# B&R Automation Studio project NAELD004C00R10L518F00 (part 43)

#### Act_Link.st
```iecst
(** 2021-05-18 **)
ACTION Act_Link:

	//ProdRcp
	bFollowerInfo	:= tyFollowerToLeaderTag.bProdWidthErr OR bProdRcpErrNotExist OR bProdRcpErrWidthMismatch;

	bLeaderInfo		:= (tyLeaderToFollowerTag.bProdWidthUSWarn OR tyLeaderToFollowerTag.bProdWidthDSWarn
	OR ((tyLeaderToFollowerTag.bProdNameUSWarn OR tyLeaderToFollowerTag.bProdNameDSWarn)
	AND (p_bAWPrep = TRUE) AND (p_bAWDis = FALSE) AND (p_eAWStat<>AWActGoWidthOff)));

	//Info Message
	IF bFollowerInfo THEN
		IF tyFollowerToLeaderTag.bProdWidthErr = TRUE OR bProdRcpErrWidthMismatch THEN

			p_sInfoMsg		:= 'Product Recipe Width Does Not Match';
			p_sInfoMsg		:= CONCAT(p_sInfoMsg , '$r$n');
			p_sInfoMsg		:= CONCAT(p_sInfoMsg , 'Check Product Width And');
			p_sInfoMsg		:= CONCAT(p_sInfoMsg , '$r$n');
			p_sInfoMsg		:= CONCAT(p_sInfoMsg , 'Leader Request Width');

		ELSIF bProdRcpErrNotExist THEN

			p_sInfoMsg		:= 'New Product Not Found';
			p_sInfoMsg		:= CONCAT(p_sInfoMsg , '$r$n');
			p_sInfoMsg		:= CONCAT(p_sInfoMsg , 'In Product Recipe List');
			p_sInfoMsg		:= CONCAT(p_sInfoMsg , '$r$n');
			p_sInfoMsg		:= CONCAT(p_sInfoMsg , 'Create New Product');
			p_sInfoMsg		:= CONCAT(p_sInfoMsg , '$r$n');
			p_sInfoMsg		:= CONCAT(p_sInfoMsg , 'In Product Setting');
		END_IF
	ELSE

		IF (tyLeaderToFollowerTag.sReqProdRcpNm<>p_tyCurrProdRcp.sRcpNm) AND (tyLeaderToFollowerTag.sReqProdRcpNm<>'')
			AND bLeaderInfo=FALSE THEN

			p_sInfoMsg		:= 'Leader Request New Recipe';
			p_sInfoMsg		:= CONCAT(p_sInfoMsg , '$r$n');
			p_sInfoMsg		:= CONCAT(p_sInfoMsg , 'Old Recipe Name : ');
			p_sInfoMsg		:= CONCAT(p_sInfoMsg , p_tyDispProdRcp.sRcpNm);
			p_sInfoMsg		:= CONCAT(p_sInfoMsg , '$r$n');
			p_sInfoMsg		:= CONCAT(p_sInfoMsg , 'Old Recipe Width : ');
			sWidthInUMTemp	:= DINT_TO_STRING(p_tyDispProdRcp.diWidthInUM / 1000);
			p_sInfoMsg		:= CONCAT(p_sInfoMsg , sWidthInUMTemp);
			p_sInfoMsg		:= CONCAT(p_sInfoMsg , '$r$n');
			p_sInfoMsg		:= CONCAT(p_sInfoMsg , 'New Recipe Name : ');
			p_sInfoMsg		:= CONCAT(p_sInfoMsg , tyLeaderToFollowerTag.sReqProdRcpNm);
			p_sInfoMsg		:= CONCAT(p_sInfoMsg , '$r$n');
			p_sInfoMsg		:= CONCAT(p_sInfoMsg , 'New Recipe Width : ');
			sWidthInUMTemp	:= DINT_TO_STRING(tyLeaderToFollowerTag.diReqProdRcpWidth / 1000);
			p_sInfoMsg		:= CONCAT(p_sInfoMsg , sWidthInUMTemp);

		ELSIF tyLeaderToFollowerTag.bProdNameUSWarn THEN
			p_sInfoMsg		:= 'US Machine Request New Recipe';
			p_sInfoMsg		:= CONCAT(p_sInfoMsg , '$r$n');
			p_sInfoMsg		:= CONCAT(p_sInfoMsg , 'Old Recipe Name : ');
			p_sInfoMsg		:= CONCAT(p_sInfoMsg , p_tyDispProdRcp.sRcpNm);
			p_sInfoMsg		:= CONCAT(p_sInfoMsg , '$r$n');
			p_sInfoMsg		:= CONCAT(p_sInfoMsg , 'Old Recipe Width : ');
			sWidthInUMTemp	:= DINT_TO_STRING(p_tyDispProdRcp.diWidthInUM / 1000); //Modify 18052021
			p_sInfoMsg		:= CONCAT(p_sInfoMsg , sWidthInUMTemp);
			p_sInfoMsg		:= CONCAT(p_sInfoMsg , '$r$n');
			p_sInfoMsg		:= CONCAT(p_sInfoMsg , 'New Recipe Name : ');
			p_sInfoMsg		:= CONCAT(p_sInfoMsg , tyLeaderToFollowerTag.sReqProdRcpNm);
			p_sInfoMsg		:= CONCAT(p_sInfoMsg , '$r$n');
			p_sInfoMsg		:= CONCAT(p_sInfoMsg , 'New Recipe Width : ');
			sWidthInUMTemp	:= DINT_TO_STRING(tyLeaderToFollowerTag.diReqProdRcpWidth / 1000);
			p_sInfoMsg		:= CONCAT(p_sInfoMsg , sWidthInUMTemp);

		ELSIF tyLeaderToFollowerTag.bProdNameDSWarn THEN
			p_sInfoMsg		:= 'Different Recipe';
			p_sInfoMsg		:= CONCAT(p_sInfoMsg , '$r$n');
			p_sInfoMsg		:= CONCAT(p_sInfoMsg , 'From DS Machine');
			p_sInfoMsg		:= CONCAT(p_sInfoMsg , '$r$n');
			p_sInfoMsg		:= CONCAT(p_sInfoMsg , 'Current Recipe Name : ');
			p_sInfoMsg		:= CONCAT(p_sInfoMsg , p_tyCurrProdRcp.sRcpNm);
			p_sInfoMsg		:= CONCAT(p_sInfoMsg , '$r$n');
			p_sInfoMsg		:= CONCAT(p_sInfoMsg , 'Current Recipe Width : ');
			sWidthInUMTemp	:= DINT_TO_STRING(p_tyCurrProdRcp.diWidthInUM2 / 1000);
			p_sInfoMsg		:= CONCAT(p_sInfoMsg , sWidthInUMTemp);

		ELSIF tyLeaderToFollowerTag.bProdWidthUSWarn THEN
			p_sInfoMsg		:= 'Product Recipe Width Does Not Match';
			p_sInfoMsg		:= CONCAT(p_sInfoMsg , '$r$n');
			p_sInfoMsg		:= CONCAT(p_sInfoMsg , 'Check Product Width And');
			p_sInfoMsg		:= CONCAT(p_sInfoMsg , '$r$n');
			p_sInfoMsg		:= CONCAT(p_sInfoMsg , 'Leader Request Width');

		ELSIF tyLeaderToFollowerTag.bProdWidthDSWarn THEN
			p_sInfoMsg		:= 'Same Recipe : ';
			p_sInfoMsg		:= CONCAT(p_sInfoMsg , p_tyDispProdRcp.sRcpNm);
			p_sInfoMsg		:= CONCAT(p_sInfoMsg , '$r$n');
			p_sInfoMsg		:= CONCAT(p_sInfoMsg , 'But Different Width');
			p_sInfoMsg		:= CONCAT(p_sInfoMsg , '$r$n');
			p_sInfoMsg		:= CONCAT(p_sInfoMsg , 'With DS Machine');
			p_sInfoMsg		:= CONCAT(p_sInfoMsg , '$r$n');
			p_sInfoMsg		:= CONCAT(p_sInfoMsg , 'Machine Outgoing Width : ');
			sWidthInUMTemp	:= DINT_TO_STRING(p_tyDispProdRcp.diWidthInUM2 / 1000);
			p_sInfoMsg		:= CONCAT(p_sInfoMsg , sWidthInUMTemp);

		END_IF
	END_IF

	//Accept New Recipe Condition (Before Loaded New Recipe)
	IF p_eLinkNtParamProjMag = LDMagDual OR p_eLinkNtParamProjMag = LDMagTriple  THEN
		p_bAccNewRcpCond	:= (p_bLinkOpsRun = TRUE)  AND (p_bLinkConvHvBrd = FALSE);
	END_IF

	//Update New Recipe Condition (After Loaded New Recipe)
	p_bUpdtNewRcpCond	:= TRUE;

	//Recipe Different
	//p_bInternalReqProdRcpDiff	:= memcmp(ADR(p_tyCurrProdRcp) , ADR(p_tyInternalReqProdRcp) , SIZEOF(p_tyCurrProdRcp)) <> 0;
	//p_bUpdtProdRcpDiff			:= memcmp(ADR(p_tyCurrProdRcp) , ADR(tyUpdtProdRcp) , SIZEOF(p_tyCurrProdRcp)) <> 0;
	//p_bRlsBrdProdRcpDiff		:= memcmp(ADR(p_tyCurrProdRcp) , ADR(tyRlsBrdProdRcpNm) , SIZEOF(p_tyCurrProdRcp)) <> 0;

	IF p_bErr THEN
		eCurrMachineStat := InError;
	ELSE
		IF p_bWarning THEN
			eCurrMachineStat := Warning;
		ELSE
			IF p_bOps THEN
				eCurrMachineStat := Run;
			ELSE
				IF p_bManual THEN
					eCurrMachineStat := Manual;
				ELSE
					eCurrMachineStat := Stop;
				END_IF
			END_IF
		END_IF
	END_IF

END_ACTION
```

#### Act_LinkEn.st
```iecst
(** 2019-04-26 **)
ACTION Act_LinkEn:

	//Link bPrep, bEn & bDis
	IF p_bLinkNtParamProjLaneBPrep = FALSE THEN
		p_bDis	:= (p_bLinkStartupRun = TRUE) OR (p_eLinkMcParamDSACommMod = McSetCommModHermes);
	ELSE
		p_bDis	:= (p_bLinkStartupRun = TRUE) OR (p_eLinkMcParamDSACommMod = McSetCommModHermes) OR (p_eLinkMcParamDSBCommMod = McSetCommModHermes);
	END_IF

END_ACTION
```

### LCS.typ
```iecst
(*2019-07-10*)
(**)
(*Action*)

TYPE
	eLCSAction :
		(
		LCSActIdle := 0,
		LCSActAddProd := 1,
		LCSActAddMultiProd := 2,
		LCSActEditProd := 3,
		LCSActEditMultiProd := 4,
		LCSActOverWriteProd := 5,
		LCSActOverWriteMultiProd := 6,
		LCSActDelProd := 7,
		LCSActDelMultiProd := 8,
		LCSActRunProd := 9,
		LCSActUploadProd := 10,
		LCSActUploadMultiProd := 11
		);
END_TYPE

(**)
(*Data*)

TYPE
	eLCSOpsStatus :
		(
		LCSOpsStatusAuto,
		LCSOpsStatusManual,
		LCSOpsStatusStop,
		LCSOpsStatusError,
		LCSOpsStatusWarning
		);
	tyLCSTagNm : 	STRUCT
		eAct : eLCSAction;
		eStat : eLCSAction;
		udiStatus : UDINT;
		sErrMsg : STRING[200];
		iIdxAct : INT;
		iIdxStat : INT;
		tyProdRcpInfo : tyProdRcpParam;
		tyCurrProdRcpParam : tyProdRcpParam;
		sCurrRcpNm : STRING[30];
		rCurrWidth : REAL;
		eCurrOpsStatus : eLCSOpsStatus;
		usiBrdStatus : USINT;
		usiMode : USINT;
		iTopToBtm : INT;
		sLastModified : STRING[80];
		bMngRcpEn : BOOL;
		bLiveData : BOOL;
		bLFEn : BOOL;
		sMcAlmMsg : STRING[255];
		bSectionLeaderEn : BOOL;
	END_STRUCT;
END_TYPE
```

### LCSLF.var
```iecst
(*2019-06-12*)
(**)
(*Action & State & Status*)
VAR
	p_LCSLFStat : UDINT;
	p_LCSLFStatus : UDINT;
	p_LCSLFStatTxt : UDINT;
END_VAR
(**)
(*Alarm*)
VAR
	p_LCSLFAlmData : UDINT;
	p_LCSLFInfoData : UDINT;
END_VAR
(**)
(*Output*)
VAR
	p_LCSLF_PLCStatus : UDINT;
	p_LCSLFChkLmt : UDINT;
	p_LCSLFAccDataMnl : UDINT;
	p_LCSLFUpdtDataMnl : UDINT;
	p_LCSLFUpdtProdRcpNm : UDINT;
	p_LCSLFUpdtProdWidth : UDINT;
	p_LCSLFMagAccOrder : UDINT;
	p_LCSLFMagOrderPos : UDINT;
END_VAR
```

### Program Logical/LCS/LCS

#### InputRef_Link.var
```iecst
(*2019-04-24*)
(**)
VAR
	p_bLinkStartupRun : REFERENCE TO BOOL;
	p_bLinkNtParamLCSLFPrep : REFERENCE TO BOOL;
	p_bLinkNtParamLCSManageRcpPrep : REFERENCE TO BOOL;
	p_bLinkNtParamLCSReqRcpPrep : REFERENCE TO BOOL;
	p_bLinkNtParamLCSLiveDatPrep : REFERENCE TO BOOL;
	p_bLinkMcParamLCSLFEn : REFERENCE TO BOOL;
	p_bLinkMcParamLCSManageRcpEn : REFERENCE TO BOOL;
	p_bLinkMcParamLCSReqRcpEn : REFERENCE TO BOOL;
	p_bLinkMcParamLCSLiveDatEn : REFERENCE TO BOOL;
END_VAR
(**)
VAR
	p_bLinkNtParamProjLaneBPrep : REFERENCE TO BOOL;
	p_tyLinkMcParamMagParamSelected : REFERENCE TO tyMagRcpParam;
END_VAR
(**)
VAR
	p_eLinkNtParamProjMag : REFERENCE TO eLDMag;
	p_bLinkPullConvHvBrd : REFERENCE TO BOOL;
	p_bLinkBffr1MagRemoved : REFERENCE TO BOOL;
	p_bLinkBffr2MagRemoved : REFERENCE TO BOOL;
	p_bLinkBffr3MagRemoved : REFERENCE TO BOOL;
END_VAR
```

#### Local.var
```iecst
(*2019-06-12*)
(**)
(*Local Action, State & Status*)
(**)
(*Local Alarm*)
VAR
	a_tyAlmText : ARRAY[10000..10099] OF tyAlmTxt := [(sAlmText:='LCS Disable'),(sAlmText:='LCS Manage Recipe Disabled'),(sAlmText:='LCS Leader Follower Disabled'),7(0),(sAlmText:='Out Of Range While Accepting New Recipe'),(sAlmText:='Out Of Range While Managing Product'),(sAlmText:='Recipe Name Empty While Adding Product'),(sAlmText:='Recipe List Full While Adding Product'),(sAlmText:='Recipe Name Exist While Adding Product'),(sAlmText:='Recipe Program Error While Adding Product'),(sAlmText:='Check Limit Error While Adding Multiple Product'),(sAlmText:='Recipe Name Empty While Adding Multiple Product'),(sAlmText:='Recipe List Full While Adding Multiple Product'),(sAlmText:='Recipe Name Exist While Adding Multiple Product'),(sAlmText:='Recipe Program Error While Adding Multiple Product'),(sAlmText:='Check Limit Error While Editing Product'),(sAlmText:='Recipe Name Empty While Editing Product'),(sAlmText:='Recipe Name Not Exist While Editing Product'),(sAlmText:='Recipe Program Error While Editing Product'),(sAlmText:='Check Limit Error While Editing Multiple Product'),(sAlmText:='Recipe Name Empty While Editing Multiple Product'),(sAlmText:='Recipe Name Not Exist While Editing Multiple Product'),(sAlmText:='Recipe Program Error While Editing Multiple Product'),(sAlmText:='Check Limit Error While Overwriting Product'),(sAlmText:='Recipe Name Empty While Overwriting Product'),(sAlmText:='Recipe List Full While Overwriting Product'),(sAlmText:='Recipe Program Error While Overwriting Product'),(sAlmText:='Check Limit Error While Overwriting Multiple Product'),(sAlmText:='Recipe Name Empty While Overwriting Multiple Product'),(sAlmText:='Recipe List Full While Overwriting Multiple Product'),(sAlmText:='Recipe Program Error While Overwriting Multiple Product'),(sAlmText:='Check Limit Error While Deleting Product'),(sAlmText:='Recipe Name Empty While Deleting Product'),(sAlmText:='Recipe Name Not Exist While Deleting Product'),(sAlmText:='Recipe Program Error While Deleting Product'),(sAlmText:='Check Limit Error While Deleting Multiple Product'),(sAlmText:='Recipe Name Empty While Deleting Multiple Product'),(sAlmText:='Recipe Name Not Exist While Deleting Multiple Product'),(sAlmText:='Recipe Program Error While Deleting Multiple Product'),(sAlmText:='Recipe Name Empty While Uploading Product'),(sAlmText:='Recipe Name Not Exist While Uploading Product'),(sAlmText:='Recipe Program Error While Uploading Product'),(sAlmText:='Get Recipe Info Error While Editing Product'),(sAlmText:='Local Recipe Is Latest Compare With LCS Recipe While Editing Product'),(sAlmText:='Local Recipe Is Latest Compare With LCS Recipe While Editing Multiple Product'),(sAlmText:='Get Recipe Info Error While Editing Multiple Product'),48(0)];
END_VAR
(**)
(*Local Output*)
VAR
	eLCSMngRcp_LCSAct : eLCSAction;
	iLCSMngRcp_LCSIdxAct : INT;
	iLCSMngRcp_LCSIdxStat : INT;
	tyLCSMngRcp_LCSProdRcpInfo : tyProdRcpParam;
	eLCSLF_LCSAct : eLCSAction;
	tyLCSLF_LCSProdRcpInfo : tyProdRcpParam;
	bChkLmtOK : BOOL;
	bChkLmtNG : BOOL;
END_VAR
(**)
(*Local Input*)
VAR
	bPrep : BOOL := TRUE;
	bEn : BOOL := TRUE;
	bDis : BOOL := FALSE;
	eLCSMngRcp_PLCStat : eLCSAction;
	udiLCSMngRcp_PLCStatus : UDINT;
	iLCSMngRcp_PLCIdxAct : INT;
	iLCSMngRcp_PLCIdxStat : INT;
	tyLCSMngRcp_PLCProdRcpInfo : tyProdRcpParam;
	eLCSLF_PLCStat : eLCSAction;
	udiLCSLF_PLCStatus : UDINT;
	bLCSMngRcpChkLmt : BOOL;
	bLCSLFChkLmt : BOOL;
	bOpsRun : BOOL;
	bError : BOOL;
	bWarning : BOOL;
	bInfo : BOOL;
	bUIManual : BOOL;
	tyProdRcpCurrRcp : tyProdRcpParam;
	tyNtParamCurr : tyNtParam;
	sProgNm : STRING[15] := 'LCS';
	bNtSettingsLoadDone : BOOL := TRUE;
END_VAR
(**)
(*Local*)
VAR
	bInitDone : BOOL;
	bInitialDone : BOOL;
	tyTagNm : tyLCSTagNm;
	bLFRun : BOOL;
	bMngRcpRun : BOOL;
	sLastModifiedTemp : STRING[80];
	sAddMsg : STRING[80];
END_VAR
```

#### Act_Background.st
```iecst
(** 2019-05-21 **)
ACTION Act_Background:

	Act_Background_LiveData;

END_ACTION
```

#### Act_InitGlobal.st
```iecst
(** 2019-06-12 **)
ACTION Act_InitGlobal:

	(* Always Change If Project Change *)

	//Pass Data To Link
	p_bLinkStartupRun ACCESS p_StartupRun;
	p_bLinkNtParamLCSLFPrep ACCESS p_NtParamLCSLFPrep;
	p_bLinkNtParamLCSManageRcpPrep ACCESS p_NtParamLCSManageRcpPrep;
	p_bLinkNtParamLCSReqRcpPrep ACCESS p_NtParamLCSReqRcpPrep;
	p_bLinkNtParamLCSLiveDatPrep ACCESS p_NtParamLCSLiveDatPrep;
	p_bLinkMcParamLCSLFEn ACCESS p_McParamLCSLFEn;
	p_bLinkMcParamLCSManageRcpEn ACCESS p_McParamLCSManageRcpEn;
	p_bLinkMcParamLCSReqRcpEn ACCESS p_McParamLCSReqRcpEn;
	p_bLinkMcParamLCSLiveDatEn ACCESS p_McParamLCSLiveDatEn;

	p_bLinkNtParamProjLaneBPrep ACCESS p_NtParamProjLaneBPrep;
	p_tyLinkMcParamMagParamSelected ACCESS p_MagRcpCurrRcp;

	p_eLinkNtParamProjMag ACCESS p_NtParamProjMag;
	p_bLinkPullConvHvBrd ACCESS p_PullConvHvBrd;
	p_bLinkBffr1MagRemoved ACCESS p_Buffer1MagRemoved;
	p_bLinkBffr2MagRemoved ACCESS p_Buffer2MagRemoved;
	p_bLinkBffr3MagRemoved ACCESS p_Buffer3MagRemoved;

	//Pass Data To Internal Use
	p_eLCSMngRcp_PLCStat ACCESS p_LCSMngRcpStat;
	p_udiLCSMngRcp_PLCStatus ACCESS p_LCSMngRcp_PLCStatus;
	p_iLCSMngRcp_PLCIdxAct ACCESS p_LCSMngRcp_PLCIdxAct;
	p_iLCSMngRcp_PLCIdxStat ACCESS p_LCSMngRcp_PLCIdxStat;
	p_tyLCSMngRcp_PLCProdRcpInfo ACCESS p_LCSMngRcp_PLCProdRcpInfo;
	p_eLCSLF_PLCStat ACCESS p_LCSLFStat;
	p_udiLCSLF_PLCStatus ACCESS p_LCSLF_PLCStatus;
	p_bLCSMngRcpChkLmt ACCESS p_LCSMngRcpChkLmt;
	p_bLCSLFChkLmt ACCESS p_LCSLFChkLmt;
	p_bOpsRun ACCESS p_OpsRun;
	p_bError ACCESS p_AlarmErr;
	p_bWarning ACCESS p_AlarmWarning;
	p_bInfo ACCESS p_AlarmInfo;
	p_bUIManual ACCESS p_UIUIMnlMod;
	p_tyProdRcpCurrRcp ACCESS p_Follower2UpdtProdRcp;	//Assign With Conveyor Last Zone (Live Data Update)
	p_tyNtParamCurr ACCESS p_NtParamCurr;
	p_sProgNm ACCESS p_NtParamLCSProgNm;
	p_bNtSettingsLoadDone ACCESS p_StartupNtSettingsLoadDone;

	(* Always Change If Project Change *)

END_ACTION
```

#### Act_Link.st
```iecst
(** 2019-07-15 **)
ACTION Act_Link:

	//Check Limit
	IF p_bLCSMngRcpChkLmt OR p_bLCSLFChkLmt THEN

		IF tyTagNm.tyProdRcpInfo.sRcpNm = '' THEN

			bChkLmtOK	:= FALSE;
			bChkLmtNG	:= TRUE;
			sAddMsg		:= 'Recipe Name Empty ';

		ELSIF tyTagNm.tyProdRcpInfo.diWidthInUM < p_tyNtParamCurr.tyProdRcpWidth.diMin THEN

			bChkLmtOK	:= FALSE;
			bChkLmtNG	:= TRUE;
			sAddMsg		:= 'Width Lower Limit ';

		ELSIF tyTagNm.tyProdRcpInfo.diWidthInUM > p_tyNtParamCurr.tyProdRcpWidth.diMax THEN

			bChkLmtOK	:= FALSE;
			bChkLmtNG	:= TRUE;
			sAddMsg		:= 'Width Upper Limit ';

		ELSIF NOT p_bLinkNtParamProjLaneBPrep AND (tyTagNm.tyProdRcpInfo.usiMcMod < DINT_TO_USINT(p_tyNtParamCurr.tyProdRcpMcModA.diMin)) THEN

			bChkLmtOK	:= FALSE;
			bChkLmtNG	:= TRUE;
			sAddMsg		:= 'Machine Mode Lower Limit ';

		ELSIF NOT p_bLinkNtParamProjLaneBPrep AND (tyTagNm.tyProdRcpInfo.usiMcMod > DINT_TO_USINT(p_tyNtParamCurr.tyProdRcpMcModA.diMax)) THEN

			bChkLmtOK	:= FALSE;
			bChkLmtNG	:= TRUE;
			sAddMsg		:= 'Machine Mode Upper Limit ';

		ELSIF p_bLinkNtParamProjLaneBPrep AND (tyTagNm.tyProdRcpInfo.usiMcMod < DINT_TO_USINT(p_tyNtParamCurr.tyProdRcpMcModAB.diMin)) THEN

			bChkLmtOK	:= FALSE;
			bChkLmtNG	:= TRUE;
			sAddMsg		:= 'Machine Mode Lower Limit ';

		ELSIF p_bLinkNtParamProjLaneBPrep AND (tyTagNm.tyProdRcpInfo.usiMcMod > DINT_TO_USINT(p_tyNtParamCurr.tyProdRcpMcModAB.diMax)) THEN

			bChkLmtOK	:= FALSE;
			bChkLmtNG	:= TRUE;
			sAddMsg		:= 'Machine Mode Upper Limit ';

		ELSIF tyTagNm.tyProdRcpInfo.diMaxSltValue < tyTagNm.tyProdRcpInfo.diMinSltValue THEN

			bChkLmtOK	:= FALSE;
			bChkLmtNG	:= TRUE;
			sAddMsg		:= 'Max Slot Lower Limit ';

		ELSIF tyTagNm.tyProdRcpInfo.diMaxSltValue > p_tyLinkMcParamMagParamSelected.diTtlSlt THEN

			bChkLmtOK	:= FALSE;
			bChkLmtNG	:= TRUE;
			sAddMsg		:= 'Max Slot Upper Limit ';

		ELSIF tyTagNm.tyProdRcpInfo.diMinSltValue < p_tyNtParamCurr.diProjMagMinSlt THEN

			bChkLmtOK	:= FALSE;
			bChkLmtNG	:= TRUE;
			sAddMsg		:= 'Min Slot Lower Limit ';

		ELSIF tyTagNm.tyProdRcpInfo.diMinSltValue > tyTagNm.tyProdRcpInfo.diMaxSltValue THEN

			bChkLmtOK	:= FALSE;
			bChkLmtNG	:= TRUE;
			sAddMsg		:= 'Min Slot Upper Limit ';

		ELSIF tyTagNm.tyProdRcpInfo.diPitch < p_tyNtParamCurr.tyProdRcpPitch.diMin THEN

			bChkLmtOK	:= FALSE;
			bChkLmtNG	:= TRUE;
			sAddMsg		:= 'Pitch Lower Limit ';

		ELSIF tyTagNm.tyProdRcpInfo.diPitch > (tyTagNm.tyProdRcpInfo.diMaxSltValue - tyTagNm.tyProdRcpInfo.diMinSltValue + 1) THEN

			bChkLmtOK	:= FALSE;
			bChkLmtNG	:= TRUE;
			sAddMsg		:= 'Pitch Upper Limit ';

		ELSIF LEN(tyTagNm.tyProdRcpInfo.sRcpNm) > 30 THEN

			bChkLmtOK	:= FALSE;
			bChkLmtNG	:= TRUE;
			sAddMsg		:= 'Recipe Name Length ';

		ELSE

			bChkLmtOK	:= TRUE;
			bChkLmtNG	:= FALSE;
			sAddMsg		:= '';

		END_IF

	ELSE

		bChkLmtOK	:= FALSE;
		bChkLmtNG	:= FALSE;

	END_IF

	//Update LCS Enable
	tyTagNm.bMngRcpEn		:= p_bLinkNtParamLCSManageRcpPrep AND p_bLinkMcParamLCSManageRcpEn;
	tyTagNm.bLFEn			:= p_bLinkNtParamLCSLFPrep AND p_bLinkMcParamLCSLFEn;
	tyTagNm.bLiveData		:= p_bLinkNtParamLCSLiveDatPrep AND p_bLinkMcParamLCSLiveDatEn;

	//tyTagNm.usiBrdStatus = 0 (Machine Empty)
	//tyTagNm.usiBrdStatus = 1 (Machine Not Empty)
	IF p_eLinkNtParamProjMag = LDMagDual THEN
		tyTagNm.usiBrdStatus	:= BOOL_TO_USINT(NOT(p_bLinkPullConvHvBrd = FALSE AND p_bLinkBffr1MagRemoved = TRUE AND p_bLinkBffr2MagRemoved = TRUE));
	ELSIF p_eLinkNtParamProjMag = LDMagTriple THEN
		tyTagNm.usiBrdStatus	:= BOOL_TO_USINT(NOT(p_bLinkPullConvHvBrd = FALSE AND p_bLinkBffr1MagRemoved = TRUE AND p_bLinkBffr2MagRemoved = TRUE AND p_bLinkBffr3MagRemoved = TRUE));
	END_IF

	//Action
	IF tyTagNm.eAct = LCSActRunProd THEN

		bLFRun		:= TRUE;
		bMngRcpRun	:= FALSE;

	ELSIF (tyTagNm.eAct = LCSActAddProd)
		OR (tyTagNm.eAct = LCSActAddMultiProd)
		OR (tyTagNm.eAct = LCSActEditProd)
		OR (tyTagNm.eAct = LCSActEditMultiProd)
		OR (tyTagNm.eAct = LCSActOverWriteProd)
		OR (tyTagNm.eAct = LCSActOverWriteMultiProd)
		OR (tyTagNm.eAct = LCSActDelProd)
		OR (tyTagNm.eAct = LCSActDelMultiProd)
		OR (tyTagNm.eAct = LCSActUploadProd)
		OR (tyTagNm.eAct = LCSActUploadMultiProd) THEN

		bLFRun		:= FALSE;
		bMngRcpRun	:= TRUE;

	ELSIF tyTagNm.eAct = LCSActIdle THEN

		bLFRun		:= FALSE;
		bMngRcpRun	:= FALSE;

	END_IF

	IF bLFRun = TRUE THEN
		eLCSLF_LCSAct			:= tyTagNm.eAct;
		tyLCSLF_LCSProdRcpInfo	:= tyTagNm.tyProdRcpInfo;

		tyLCSLF_LCSProdRcpInfo.bTopToBtm	:= INT_TO_BOOL(tyTagNm.iTopToBtm);

		sLastModifiedTemp	:= CONCAT('DT#' , tyTagNm.sLastModified);
		tyLCSLF_LCSProdRcpInfo.dtLastModified	:= STRING_TO_DT(sLastModifiedTemp);

		tyTagNm.eStat		:= p_eLCSLF_PLCStat;
		tyTagNm.udiStatus	:= p_udiLCSLF_PLCStatus;

		IF tyTagNm.udiStatus > 0 AND tyTagNm.udiStatus < 65534 THEN
			tyTagNm.sErrMsg	:= a_tyAlmText[tyTagNm.udiStatus].sAlmText;

			IF tyTagNm.udiStatus = 10010 OR tyTagNm.udiStatus = 10011 THEN
				tyTagNm.sErrMsg	:= CONCAT(sAddMsg , tyTagNm.sErrMsg);
			END_IF
		END_IF

	ELSIF bMngRcpRun = TRUE THEN
		eLCSMngRcp_LCSAct	:= tyTagNm.eAct;

		tyTagNm.eStat		:= p_eLCSMngRcp_PLCStat;
		tyTagNm.udiStatus	:= p_udiLCSMngRcp_PLCStatus;

		IF tyTagNm.udiStatus > 0 AND tyTagNm.udiStatus < 65534 THEN
			tyTagNm.sErrMsg	:= a_tyAlmText[tyTagNm.udiStatus].sAlmText;

			IF tyTagNm.udiStatus = 10010 OR tyTagNm.udiStatus = 10011 THEN
				tyTagNm.sErrMsg	:= CONCAT(sAddMsg , tyTagNm.sErrMsg);
			END_IF
		END_IF

		IF tyTagNm.eAct = LCSActUploadProd THEN
			IF tyTagNm.udiStatus = 0 THEN
				tyTagNm.tyProdRcpInfo	:= p_tyLCSMngRcp_PLCProdRcpInfo;

				tyTagNm.iTopToBtm	:= BOOL_TO_INT(tyLCSMngRcp_LCSProdRcpInfo.bTopToBtm);

				tyTagNm.sLastModified	:= DT_TO_STRING(tyLCSMngRcp_LCSProdRcpInfo.dtLastModified);
				tyTagNm.sLastModified	:= RIGHT(tyTagNm.sLastModified , (LEN(tyTagNm.sLastModified) - 3));

			ELSE
				tyLCSMngRcp_LCSProdRcpInfo	:= tyTagNm.tyProdRcpInfo;

				tyLCSMngRcp_LCSProdRcpInfo.bTopToBtm	:= INT_TO_BOOL(tyTagNm.iTopToBtm);
				tyLCSMngRcp_LCSProdRcpInfo.diWidthInUM2 := tyTagNm.tyProdRcpInfo.diWidthInUM;

				sLastModifiedTemp	:= CONCAT('DT#' , tyTagNm.sLastModified);
				tyLCSMngRcp_LCSProdRcpInfo.dtLastModified	:= STRING_TO_DT(sLastModifiedTemp);

			END_IF

		ELSIF tyTagNm.eAct = LCSActUploadMultiProd THEN
			iLCSMngRcp_LCSIdxStat	:= tyTagNm.iIdxAct;

			tyTagNm.iIdxStat		:= p_iLCSMngRcp_PLCIdxAct;

			tyTagNm.tyProdRcpInfo	:= p_tyLCSMngRcp_PLCProdRcpInfo;

			tyTagNm.iTopToBtm	:= BOOL_TO_INT(tyLCSMngRcp_LCSProdRcpInfo.bTopToBtm);

			tyTagNm.sLastModified	:= DT_TO_STRING(tyLCSMngRcp_LCSProdRcpInfo.dtLastModified);
			tyTagNm.sLastModified	:= RIGHT(tyTagNm.sLastModified , (LEN(tyTagNm.sLastModified) - 3));

		ELSE
			iLCSMngRcp_LCSIdxAct		:= tyTagNm.iIdxAct;
			tyLCSMngRcp_LCSProdRcpInfo	:= tyTagNm.tyProdRcpInfo;

			tyLCSMngRcp_LCSProdRcpInfo.bTopToBtm	:= INT_TO_BOOL(tyTagNm.iTopToBtm);
			tyLCSMngRcp_LCSProdRcpInfo.diWidthInUM2 := tyTagNm.tyProdRcpInfo.diWidthInUM;

			sLastModifiedTemp	:= CONCAT('DT#' , tyTagNm.sLastModified);
			tyLCSMngRcp_LCSProdRcpInfo.dtLastModified	:= STRING_TO_DT(sLastModifiedTemp);

			tyTagNm.iIdxStat	:= p_iLCSMngRcp_PLCIdxStat;

		END_IF

	ELSE

		eLCSLF_LCSAct		:= LCSActIdle;
		eLCSMngRcp_LCSAct	:= LCSActIdle;
		tyTagNm.eStat		:= LCSActIdle;
		tyTagNm.udiStatus	:= 65534;
		tyTagNm.sErrMsg		:= '';

	END_IF

END_ACTION
```

#### Init.st
```iecst
(** 2019-04-24 **)
PROGRAM _INIT

	(* Always Change If Project Change *)

	//Pass Address To Global Address For External Use
	//Action, State & Status

	//Alarm

	//Output
	p_LCS_LCSMngRcp_LCSAct			:= ADR(eLCSMngRcp_LCSAct);
	p_LCS_LCSMngRcp_LCSIdxAct		:= ADR(iLCSMngRcp_LCSIdxAct);
	p_LCS_LCSMngRcp_LCSIdxStat		:= ADR(iLCSMngRcp_LCSIdxStat);
	p_LCS_LCSMngRcp_LCSProdRcpInfo	:= ADR(tyLCSMngRcp_LCSProdRcpInfo);
	p_LCS_LCSLF_LCSAct				:= ADR(eLCSLF_LCSAct);
	p_LCS_LCSLF_LCSProdRcpInfo		:= ADR(tyLCSLF_LCSProdRcpInfo);
	p_LCSChkLmtOK					:= ADR(bChkLmtOK);
	p_LCSChkLmtNG					:= ADR(bChkLmtNG);
	p_LCSSectionLeaderEn			:= ADR(tyTagNm.bSectionLeaderEn);

	(* Always Change If Project Change *)

END_PROGRAM
```

### Program Logical/LCS/LCSLF

#### InputRef_Link.var
```iecst
(*2019-04-24*)
(**)
VAR
	sWidthInUMTemp : STRING[80];
	p_bLinkStartupRun : REFERENCE TO BOOL;
END_VAR
(**)
VAR
	p_bLinkNtParamProjLaneBPrep : REFERENCE TO BOOL;
	p_eLinkMcParamDSACommMod : REFERENCE TO eMcSetCommMod;
	p_eLinkMcParamDSBCommMod : REFERENCE TO eMcSetCommMod;
END_VAR
(**)
VAR
	p_bLinkOpsRun : REFERENCE TO BOOL;
	p_bLinkConvHvBrd : REFERENCE TO BOOL;
	p_bLinkOpsMagConvLD1QueryWO : REFERENCE TO BOOL;
	p_bLinkOpsMagConvLD2QueryWO : REFERENCE TO BOOL;
	p_bLinkOpsMagConvLD3QueryWO : REFERENCE TO BOOL;
	p_tyDTStructure : REFERENCE TO DTStructure;
	p_tyResponseFromMES1 : REFERENCE TO tyStatPlatformFromMES;
	p_tyResponseFromMES2 : REFERENCE TO tyStatPlatformFromMES;
	p_tyResponseFromMES3 : REFERENCE TO tyStatPlatformFromMES;
END_VAR
```

#### Local.var
```iecst
(*2019-06-28*)
(**)
(*Local Action, State & Status*)
VAR
	eAct : eLCSAction := LCSActIdle;
	eStat : eLCSAction := LCSActIdle;
	eStatus : eFBStatus := Idle;
	udiStatus : UDINT := 0;
	sStatTxt : STRING[200] := '';
	a_sStatText : ARRAY[0..50] OF STRING[200] := ['Idling','Adding Product','Adding Multiple Products','Editing Product','Editing Multiple Products','OverWrite Product','OverWrite Multiple Products','Deleting Product','Deleting Multiple Products','Running LCS Product','Uploading Product','Uploading Multiple Products',39('')];
END_VAR
(**)
(*Local Alarm*)
VAR
	tyAlmData : tyAlmDat;
	tyInfoData : tyAlmDat;
	a_tyAlmText : ARRAY[10000..10099] OF tyAlmTxt;
END_VAR
(**)
(*Local Output*)
VAR
	udiPLCStatus : UDINT;
	bChkLmt : BOOL;
	bAccDataMnl : BOOL;
	bUpdtDataMnl : BOOL;
	sUpdtProdRcpNm : STRING[30];
	diUpdtProdWidth : DINT;
END_VAR
(**)
(*Local Input*)
VAR
	udiRstErr : UDINT := 0;
	bPrep : BOOL := TRUE;
	bEn : BOOL := TRUE;
	bDis : BOOL := FALSE;
	tyCurrProdParam : tyProdRcpParam;
	bMnlAccData : BOOL;
	bAccData : BOOL;
	tyLCSProdRcpInfo : tyProdRcpParam;
	bChkLmtOK : BOOL;
	bChkLmtNG : BOOL;
	bAccNewRcpCond : BOOL;
	bUpdtNewRcpCond : BOOL;
	bAutoUpdtData : BOOL;
	bUIUpdtData : BOOL;
	sInfoMsg : STRING[200];
	sProgNm : STRING[15] := 'LCSLF';
	bNtSettingsLoadDone : BOOL := TRUE;
END_VAR
(**)
(*Local*)
VAR
	bRstErr : BOOL;
	udiRstErrOld : UDINT;
	bInitDone : BOOL;
	bInitialDone : BOOL;
	usiStep : USINT;
	usiProdUpdtDatStep : USINT;
	udiModuleNum : UDINT := 4101;
END_VAR
(*Local priority param*)
VAR
	bGUIDInserted : ARRAY[1..3] OF BOOL;
	a_MagGUID : ARRAY[1..3] OF STRING[80];
END_VAR
VAR RETAIN
	a_MagAccOrder : ARRAY[1..3] OF USINT; (*priority (output)*)
END_VAR
VAR
	usiMagPrior : ARRAY[1..3] OF USINT := [1,2,3];
	usiMagRun : ARRAY[1..3] OF USINT;
	usiSum : ARRAY[1..3] OF USINT;
	usiMagOrderPos : USINT;
	i : USINT;
	i1 : USINT;
	uiMilliSecOld : UINT;
END_VAR
```

#### Act_Alarm.st
```iecst
(** 2019-04-24 **)
ACTION Act_Alarm:

	//Error
	IF EDGEPOS(eStatus = Error) THEN

		tyAlmData.sProgNm		:= p_sProgNm;
		tyAlmData.udiCode		:= udiStatus;
		tyAlmData.eSeverity		:= AlmSeverityError;
		tyAlmData.udiRunTime	:= tyAlmData.udiRunTime + 1;
		tyAlmData.bAlm			:= TRUE;
		tyAlmData.udiModuleNum  := udiModuleNum;
		g_sLCSLFProgNm			:= p_sProgNm;

		//Get Error Message
		IF tyAlmData.udiCode < 10000 OR tyAlmData.udiCode > 10099 THEN
			tyAlmData.sAlmMsg	:= 'Unknown';
			tyAlmData.sRcyMsg	:= 'Unknown';
		ELSE
			tyAlmData.sAlmMsg	:= a_tyAlmText[tyAlmData.udiCode].sAlmText;
			tyAlmData.sRcyMsg	:= a_tyAlmText[tyAlmData.udiCode].sRcyText;
		END_IF

		sStatTxt	:= tyAlmData.sAlmMsg;

	ELSIF bRstErr AND (tyAlmData.udiCode <> 0) THEN

		tyAlmData.udiCode	:= 0;
		tyAlmData.eSeverity	:= AlmSeverityNA;
		tyAlmData.sAlmMsg	:= '';
		tyAlmData.sRcyMsg	:= '';
		tyAlmData.bAlm			:= FALSE;
		sStatTxt	:= a_sStatText[eStat];

	END_IF

END_ACTION
```

#### Act_InitGlobal.st
```iecst
(** 2019-05-07 **)
ACTION Act_InitGlobal:

	(* Always Change If Project Change *)

	//Pass Data To Link
	p_bLinkStartupRun ACCESS p_StartupRun;
	p_bLinkNtParamProjLaneBPrep ACCESS p_NtParamProjLaneBPrep;
	p_eLinkMcParamDSACommMod ACCESS p_McParamDSCommAMod;
	p_eLinkMcParamDSBCommMod ACCESS p_McParamDSCommBMod;

	p_bLinkOpsRun ACCESS p_OpsRun;
	p_bLinkConvHvBrd ACCESS p_PullConvHvBrd;
	p_bLinkOpsMagConvLD1QueryWO ACCESS p_OpsMagConvLD1QueryWO;
	p_bLinkOpsMagConvLD2QueryWO ACCESS p_OpsMagConvLD2QueryWO;
	p_bLinkOpsMagConvLD3QueryWO ACCESS p_OpsMagConvLD3QueryWO;
	p_tyDTStructure ACCESS p_TimeCurrDTStruct;
	p_tyResponseFromMES1 ACCESS p_TagFromMesMagConv1; //For we_fab
	p_tyResponseFromMES2 ACCESS p_TagFromMesMagConv2; //For we_fab
	p_tyResponseFromMES3 ACCESS p_TagFromMesMagConv3; //For we_fab

	//Pass Data To Internal Use
	p_eAct ACCESS p_LCS_LCSLF_LCSAct;
	p_udiRstErr ACCESS p_RstErrReset;
	p_bPrep ACCESS p_NtParamLCSLFPrep;
	p_bEn ACCESS p_McParamLCSLFEn;
	p_tyCurrProdParam ACCESS p_ProdRcpCurrRcp0;
	p_bMnlAccData ACCESS p_McParamMnlAccDat;
	p_bAccData ACCESS p_UIProdAccData;
	p_tyLCSProdRcpInfo ACCESS p_LCS_LCSLF_LCSProdRcpInfo;
	p_bChkLmtOK ACCESS p_LCSChkLmtOK;
	p_bChkLmtNG ACCESS p_LCSChkLmtNG;
	p_sProgNm ACCESS p_NtParamLCSLFProgNm;
	p_bNtSettingsLoadDone ACCESS p_StartupNtSettingsLoadDone;

	p_bUIBtnSectionLdr ACCESS P_UISectionLdr;
	p_bLCSSectionLeaderEn ACCESS p_LCSSectionLeaderEn;
	p_bMcParamSectionLdr ACCESS p_McParamSectionLeader;

	(* Always Change If Project Change *)

END_ACTION
```

#### Act_Link.st
```iecst
(** 2019-06-28 **)
ACTION Act_Link:

	p_sInfoMsg		:= 'LCS Request New Recipe';
	p_sInfoMsg		:= CONCAT(p_sInfoMsg , '$r$n');
	p_sInfoMsg		:= CONCAT(p_sInfoMsg , 'Old Recipe Name : ');
	p_sInfoMsg		:= CONCAT(p_sInfoMsg , p_tyCurrProdParam.sRcpNm);
	p_sInfoMsg		:= CONCAT(p_sInfoMsg , '$r$n');
	p_sInfoMsg		:= CONCAT(p_sInfoMsg , 'Old Recipe Width : ');
	sWidthInUMTemp	:= DINT_TO_STRING(p_tyCurrProdParam.diWidthInUM / 1000);
	p_sInfoMsg		:= CONCAT(p_sInfoMsg , sWidthInUMTemp);
	p_sInfoMsg		:= CONCAT(p_sInfoMsg , '$r$n');
	p_sInfoMsg		:= CONCAT(p_sInfoMsg , 'New Recipe Name : ');
	p_sInfoMsg		:= CONCAT(p_sInfoMsg , p_tyLCSProdRcpInfo.sRcpNm);
	p_sInfoMsg		:= CONCAT(p_sInfoMsg , '$r$n');
	p_sInfoMsg		:= CONCAT(p_sInfoMsg , 'New Recipe Width : ');
	sWidthInUMTemp	:= DINT_TO_STRING(p_tyLCSProdRcpInfo.diWidthInUM / 1000);
	p_sInfoMsg		:= CONCAT(p_sInfoMsg , sWidthInUMTemp);

	//Accept New Recipe Condition
	p_bAccNewRcpCond	:= p_bLinkOpsRun = TRUE AND p_bLinkConvHvBrd = FALSE;

	//@@@@@@@@@@@@@@@@@@@@@@@@@@@@@@@@@@@@@@@@@@@@@@@@@@@@@@@@@@@@@@@@@@@@@@
	//we_fabricate
//	IF  uiMilliSecOld <> p_tyDTStructure.millisec THEN
//		IF EDGEPOS(p_bLinkOpsMagConvLD1QueryWO) THEN //query false when rcp loaded
//			sMagazineId 		:= '1'; //Magazine position to mes
//			bGUIDInserted[1]	:= FALSE;
//			a_bQueryQueue[i2] 	:= TRUE;
//			i2 := i2 + 1;
//		ELSIF EDGEPOS(p_bLinkOpsMagConvLD2QueryWO) THEN
//			sMagazineId 		:= '2';
//			bGUIDInserted[2]	:= FALSE;
//			a_bQueryQueue[i2] 	:= TRUE;
//			i2 := i2 + 1;
//		ELSIF EDGEPOS(p_bLinkOpsMagConvLD3QueryWO) THEN
//			sMagazineId 		:= '3';
//			bGUIDInserted[3]	:= FALSE;
//			a_bQueryQueue[i2] 	:= TRUE;
//			i2 := i2 + 1;
//		END_IF
//	END_IF
	IF  uiMilliSecOld <> p_tyDTStructure.millisec THEN
		//Priority setting
		IF EDGEPOS(p_tyResponseFromMES1.iAcceptCondition >0)  OR EDGEPOS(p_tyResponseFromMES2.iAcceptCondition > 0)  OR EDGEPOS(p_tyResponseFromMES3.iAcceptCondition >0) THEN
			uiMilliSecOld :=  p_tyDTStructure.millisec;
			memset(ADR(usiSum),0,SIZEOF(usiSum));
			IF p_tyResponseFromMES1.iAcceptCondition >0 THEN
				usiSum[1] := 11;
			ELSIF p_tyResponseFromMES2.iAcceptCondition >0 THEN
				usiSum[2] := 12;
			ELSIF p_tyResponseFromMES3.iAcceptCondition >0 THEN
				usiSum[3] := 13;
			END_IF
		ELSE
			memset(ADR(usiSum),0,SIZEOF(usiSum));
		END_IF
	END_IF

//	FOR i := 1 TO 3 DO
//		usiSum[i]	:= usiSum[i] + usiMagPrior[i];
//		IF a_MagGUID[i] = tySendWorkOrderInfoRcv.tyData.sQueryId THEN
//			usiSum[i] := usiSum[i] + 10;
//		END_IF
//	END_FOR

	FOR i1:=1 TO 3 DO
		//Assign Magazine order
		IF  usiSum[i1] >=10 THEN
			IF a_MagAccOrder[1]=0 AND a_MagAccOrder[2]=0 AND a_MagAccOrder[3]=0 THEN
				a_MagAccOrder[i1] := 10; //output
				usiMagOrderPos := i1;
			ELSIF ((a_MagAccOrder[1]=0 AND a_MagAccOrder[2]=0) OR
				(a_MagAccOrder[2]=0 AND a_MagAccOrder[3]=0) OR
				(a_MagAccOrder[1]=0 AND a_MagAccOrder[3]=0)) AND a_MagAccOrder[i1] =0 THEN
				a_MagAccOrder[i1] := 20;
				usiMagOrderPos := i1;
			ELSIF (a_MagAccOrder[1]=0 OR a_MagAccOrder[2]=0 OR a_MagAccOrder[3]=0) AND a_MagAccOrder[i1] =0 THEN
				a_MagAccOrder[i1] := 30;
				usiMagOrderPos := i1;
			END_IF
			bGUIDInserted[i1] := FALSE;
		END_IF
	END_FOR

	//update magazine mmy
	IF a_MagAccOrder[1]<>0 AND a_MagAccOrder[2]<>0 AND a_MagAccOrder[3]<>0 THEN
	ELSIF a_MagAccOrder[1]<>10 AND a_MagAccOrder[2]<>10 AND a_MagAccOrder[3]<>10 THEN
		FOR i := 1 TO 3 DO
			IF a_MagAccOrder[i] <> 0 THEN
				a_MagAccOrder[i] := a_MagAccOrder[i] -10;
			END_IF
		END_FOR
	END_IF

END_ACTION
```

#### Act_LinkEn.st
```iecst
(** 2019-04-24 **)
ACTION Act_LinkEn:

	//Link bPrep, bEn & bDis
	IF p_bLinkNtParamProjLaneBPrep = FALSE THEN
		p_bDis	:= (p_bLinkStartupRun = TRUE) OR (p_eLinkMcParamDSACommMod = McSetCommModHermes);
	ELSE
		p_bDis	:= (p_bLinkStartupRun = TRUE) OR (p_eLinkMcParamDSACommMod = McSetCommModHermes) OR (p_eLinkMcParamDSBCommMod = McSetCommModHermes);
	END_IF

END_ACTION
```

#### Act_Main.st
```iecst
(** 2019-06-28 **)
ACTION Act_Main:

	//Main
	CASE eStat OF

		LCSActIdle:
			IF eStatus <> Idle THEN	//Reset Data
				//Private
				usiStep		:= 0;
				bAccDataMnl	:= FALSE;
				bChkLmt		:= FALSE;

				tyInfoData.sProgNm		:= '';
				tyInfoData.udiCode		:= 0;
				tyInfoData.eSeverity	:= AlmSeverityNA;
				tyInfoData.sAlmMsg		:= '';

				sStatTxt	:= a_sStatText[eStat];

			END_IF

			eStatus			:= Idle;
			udiPLCStatus	:= 65534;

		LCSActRunProd:
			IF eStatus = Idle OR eStatus = Busy THEN

				eStatus			:= Busy;
				udiPLCStatus	:= 65535;

				sStatTxt	:= a_sStatText[eStat];

				CASE usiStep OF
					0:
						//Check Limit
						bChkLmt	:= TRUE;

						IF p_bChkLmtOK = TRUE THEN
							usiStep			:= 1;
						ELSIF p_bChkLmtNG = TRUE THEN
							eStatus			:= Done;
							udiPLCStatus	:= 10010;	//Out Of Range While Accepting New Recipe
						END_IF

					1:
						//Manual Accept Data Check
						IF p_bMnlAccData = TRUE THEN
							bAccDataMnl	:= TRUE;

							//Info Message
							tyInfoData.sProgNm		:= p_sProgNm;
							tyInfoData.udiCode		:= 10000;
							tyInfoData.eSeverity	:= AlmSeverityInfo;
							tyInfoData.sAlmMsg		:= p_sInfoMsg;

							IF p_bAccData = TRUE THEN
								p_bAccData := FALSE; //2023_07_26_Debug for Manual Accept Data automatically accept after product change many times
								bAccDataMnl	:= FALSE;
								usiStep		:= 2;
							END_IF
						ELSE
							p_bAccData := FALSE; //2023_07_26_Debug for Manual Accept Data automatically accept after product change many times
							bAccDataMnl	:= FALSE;
							usiStep		:= 2;
						END_IF

					2:
						//Accept New Recipe Condition
						IF p_bAccNewRcpCond = TRUE THEN
							usiStep	:= 3;
						ELSE
							//Info Message
							tyInfoData.sProgNm		:= p_sProgNm;
							tyInfoData.udiCode		:= 10000;
							tyInfoData.eSeverity	:= AlmSeverityInfo;
							tyInfoData.sAlmMsg		:= p_sInfoMsg;
						END_IF

					3:
						//Accept New Recipe
						p_tyCurrProdParam	:= p_tyLCSProdRcpInfo;

						IF p_bLCSSectionLeaderEn = TRUE THEN
							p_bMcParamSectionLdr	:= TRUE;
							p_bUIBtnSectionLdr		:= TRUE;
						ELSE
							p_bMcParamSectionLdr	:= FALSE;
							p_bUIBtnSectionLdr		:= FALSE;

						END_IF

						usiStep	:= 4;

					4:
						//Clear Info Message
						tyInfoData.sProgNm		:= '';
						tyInfoData.udiCode		:= 0;
						tyInfoData.eSeverity	:= AlmSeverityNA;
						tyInfoData.sAlmMsg		:= '';

						usiStep	:= 0;

						eStatus			:= Done;
						udiPLCStatus	:= 0;

				END_CASE

			END_IF

		ELSE
			IF eStatus = Idle OR eStatus = Busy THEN
				eStatus	:= Done;
			END_IF

	END_CASE

END_ACTION
```

#### Init.st
```iecst
(** 2019-06-12 **)
PROGRAM _INIT

	(* Always Change If Project Change *)

	//Pass Address To Global Address For External Use
	//Action, State & Status
	p_LCSLFStat		:= ADR(eStat);
	p_LCSLFStatus	:= ADR(eStatus);
	p_LCSLFStatTxt	:= ADR(sStatTxt);

	//Alarm
	p_LCSLFAlmData	:= ADR(tyAlmData);
	p_LCSLFInfoData	:= ADR(tyInfoData);

	//Output
	p_LCSLF_PLCStatus		:= ADR(udiPLCStatus);
	p_LCSLFChkLmt			:= ADR(bChkLmt);
	p_LCSLFAccDataMnl		:= ADR(bAccDataMnl);
	p_LCSLFUpdtDataMnl		:= ADR(bUpdtDataMnl);
	p_LCSLFUpdtProdRcpNm	:= ADR(sUpdtProdRcpNm);
	p_LCSLFUpdtProdWidth	:= ADR(diUpdtProdWidth);

	p_LCSLFMagAccOrder 			:= ADR(a_MagAccOrder);
	p_LCSLFMagOrderPos 			:= ADR(usiMagOrderPos);

	(* Always Change If Project Change *)

END_PROGRAM
```

### Program Logical/LCS/LCSMngRcp

#### Act_Alarm.st
```iecst
(** 2019-04-24 **)
ACTION Act_Alarm:

	//Error
	IF EDGEPOS(eStatus = Error) THEN

		tyAlmData.sProgNm		:= p_sProgNm;
		tyAlmData.udiCode		:= udiStatus;
		tyAlmData.eSeverity		:= AlmSeverityError;
		tyAlmData.udiRunTime	:= tyAlmData.udiRunTime + 1;
		tyAlmData.bAlm			:= TRUE;
		tyAlmData.udiModuleNum  := udiModuleNum;
		g_sLCSMngRcpProgNm		:= p_sProgNm;

		//Get Error Message
		IF tyAlmData.udiCode < 10000 OR tyAlmData.udiCode > 10099 THEN
			tyAlmData.sAlmMsg	:= 'Unknown';
			tyAlmData.sRcyMsg	:= 'Unknown';
		ELSE
			tyAlmData.sAlmMsg	:= a_tyAlmText[tyAlmData.udiCode].sAlmText;
			tyAlmData.sRcyMsg	:= a_tyAlmText[tyAlmData.udiCode].sRcyText;
		END_IF

		sStatTxt	:= tyAlmData.sAlmMsg;

	ELSIF bRstErr AND (tyAlmData.udiCode <> 0) THEN

		tyAlmData.udiCode	:= 0;
		tyAlmData.eSeverity	:= AlmSeverityNA;
		tyAlmData.sAlmMsg	:= '';
		tyAlmData.sRcyMsg	:= '';
		tyAlmData.bAlm			:= FALSE;
		sStatTxt	:= a_sStatText[eStat];

	END_IF

END_ACTION
```

### Program Logical/Operations/Ops (IEC) - 1.00.0 - 

#### InputRef_Link.var
```iecst
(*2019-01-20*)
(**)
(*External*)
VAR
	p_bLinkOpsTravLifLDPaused : REFERENCE TO BOOL;
	p_bLinkOpsMagLD1Paused : REFERENCE TO BOOL;
	p_bLinkOpsMagLD2Paused : REFERENCE TO BOOL;
	p_bLinkOpsMagLD3Paused : REFERENCE TO BOOL;
	p_bLinkOpsMagLD4Paused : REFERENCE TO BOOL;
	p_bLinkOpsMagConvLD1Paused : REFERENCE TO BOOL;
	p_bLinkOpsMagConvLD2Paused : REFERENCE TO BOOL;
	p_bLinkOpsMagConvLD3Paused : REFERENCE TO BOOL;
	p_bLinkOpsMagConvLD4Paused : REFERENCE TO BOOL;
	p_bLinkUIOpsAct : REFERENCE TO eOperationsAction;
	p_bLinkSimuRun : REFERENCE TO BOOL;
	p_bLinkSimuStop : REFERENCE TO BOOL;
	p_bLinkOpsLifMagLDPaused : REFERENCE TO BOOL;
	p_bLinkProjLifterMagPlatform : REFERENCE TO BOOL;
END_VAR
```

#### Act_InitGlobal.st
```iecst
(** 2019-03-22 **)
ACTION Act_InitGlobal:

	(* Always Change If Project Change *)

	//Pass Data To Link
	p_bLinkOpsTravLifLDPaused ACCESS p_OpsTravLifLDPaused;
//	p_bLinkOpsMagLD1Paused ACCESS p_OpsMagLD1Paused;
//	p_bLinkOpsMagLD2Paused ACCESS p_OpsMagLD2Paused;
//	p_bLinkOpsMagLD3Paused ACCESS p_OpsMagLD3Paused;
//	p_bLinkOpsMagLD4Paused ACCESS p_OpsMagLD4Paused;
	p_bLinkOpsMagConvLD1Paused ACCESS p_OpsMagConvLD1Paused;
	p_bLinkOpsMagConvLD2Paused ACCESS p_OpsMagConvLD2Paused;
	p_bLinkOpsMagConvLD3Paused ACCESS p_OpsMagConvLD3Paused;
	p_bLinkOpsMagConvLD4Paused ACCESS p_OpsMagConvLD4Paused;
	p_bLinkUIOpsAct ACCESS p_UIOpsAct;
	p_bLinkSimuRun ACCESS p_SimuRun;
	p_bLinkSimuStop ACCESS p_SimuStop;

	p_bLinkProjLifterMagPlatform ACCESS p_NtParamProjLifterMagPlatform;
	p_bLinkOpsLifMagLDPaused ACCESS p_OpsLifMagLDPaused;

	//Pass Data To Internal Use
//	p_eAct ACCESS p_UIOpsAct;
	p_udiRstErr ACCESS p_RstErrReset;
	p_bNtSettingsLoadDone ACCESS p_StartupNtSettingsLoadDone;

	(* Always Change If Project Change *)

END_ACTION
```

#### Act_Link.st
```iecst
(** 2019-01-20 **)
ACTION Act_Link:

	IF p_bLinkProjLifterMagPlatform THEN

		p_bPaused	:= 	(p_bLinkOpsTravLifLDPaused AND p_bLinkOpsLifMagLDPaused);

	ELSE

		p_bPaused	:= 	(p_bLinkOpsTravLifLDPaused
	//					AND p_bLinkOpsMagLD1Paused AND p_bLinkOpsMagLD2Paused AND p_bLinkOpsMagLD3Paused AND p_bLinkOpsMagLD4Paused
						AND p_bLinkOpsMagConvLD1Paused AND p_bLinkOpsMagConvLD2Paused AND p_bLinkOpsMagConvLD3Paused  AND p_bLinkOpsMagConvLD4Paused);

	END_IF

END_ACTION
```

#### Act_LinkAction.st
```iecst
(** 2019-03-29 **)
ACTION Act_LinkAction:

	IF p_bLinkUIOpsAct <> OperationsActIdle THEN
		p_eAct ACCESS p_UIOpsAct;
	ELSIF EDGEPOS(p_bLinkSimuRun) THEN
		p_eAct := OperationsActStart;
	ELSIF EDGEPOS(p_bLinkSimuStop) THEN
		p_eAct := OperationsActStop;
	END_IF

	IF (eStat = OperationsActStart OR eStat = OperationsActStop) AND  eStatus = Done THEN
		eAct := OperationsActIdle;
		p_eAct := OperationsActIdle;
	END_IF

END_ACTION
```

#### Init.st
```iecst
(** 2019-04-16 **)
PROGRAM _INIT

	(* Always Change If Project Change *)

	//Pass Address To Global Address For External Use
	//Action, State & Status
	p_OpsStat		:= ADR(eStat);
	p_OpsStatus		:= ADR(eStatus);
	p_OpsStatTxt	:= ADR(sStatTxt);

	//Alarm

	//Output
	p_OpsOpsStatus			:= ADR(eOpsStatus);
	p_OpsStatusRun			:= ADR(bStatusRun);
	p_OpsStatusStop			:= ADR(bStatusStop);
	p_OpsStatusCycleStop	:= ADR(bStatusCycleStop);
	p_OpsStatusStep			:= ADR(bStatusStep);
	p_OpsRun				:= ADR(bRun);
	p_OpsStop				:= ADR(bStop);
	p_OpsStep				:= ADR(bStep);
	p_OpsPause				:= ADR(bPaused);
	(* Always Change If Project Change *)

END_PROGRAM
```

### OpsTravLifLD.typ - Do Not Change!!!
```iecst
(*2018-12-11*)
(**)
(*Configuration*)

TYPE
	eLDMod :
		(
		LDModLoadLnA,
		LDModLoadLnB,
		LDModLoadLnAB
		);
	eLDMag :
		(
		LDMagDual,
		LDMagTriple,
		LDMagQuadruple
		);
END_TYPE

(**)

TYPE
	tyParamTravLifLD : 	STRUCT
		a_bUSDis : ARRAY[1..4]OF BOOL := [4(FALSE)];
		a_bDSDis : ARRAY[1..4]OF BOOL := [4(FALSE)];
		a_usiUSPriority : ARRAY[1..4]OF USINT := [1,2,3,1(0)];
		a_usiDSPriority : ARRAY[1..4]OF USINT := [1,2,3,1(0)];
	END_STRUCT;
END_TYPE

(**)
(*Sequence*)

TYPE
	eTravLifLDStep :
		(
		TravLifLDStepNA,
		TravLifLDStepInitConv,
		TravLifLDStepInitInletPneuCls,
		TravLifLDStepInitInOutPneuCls,
		TravLifLDStepInitTravLif,
		TravLifLDStepInitAWTravLif,
		TravLifLDStepAWMov,
		TravLifLDStepTravLifMov,
		TravLifLDStepUSSigWait,
		TravLifLDStepUSSigRechk,
		TravLifLDStepInletPneuOpn,
		TravLifLDStepUSSigRechkTwice,
		TravLifLDStepUSComm,
		TravLifLDStepEntBrd,
		TravLifLDStepInletPneuCls,
		TravLifLDStepDSSigWait,
		TravLifLDStepDSSigRechk,
		TravLifLDStepOutletPneuOpn,
		TravLifLDStepDSSigRechkTwice,
		TravLifLDStepChkRgtSenForDBAOn,
		TravLifLDStepDSComm,
		TravLifLDStepExitBrd,
		TravLifLDStepOutletPneuCls,
		TravLifLDStepTranInErr
		);
	eTravLifLDStep1 :
		(
		TravLifLDStep1NA,
		TravLifLDStep1InitConv,
		TravLifLDStep1InitInletPneuCls,
		TravLifLDStep1InitInOutPneuCls,
		TravLifLDStep1InitTravLif,
		TravLifLDStep1InitAWTravLif,
		TravLifLDStep1DSSigWait100,
		TravLifLDStep1AWMov,
		TravLifLDStep1Standby,
		TravLifLDStep1USSigWait,
		TravLifLDStep1PreEntAllServo200,
		TravLifLDStep1PreEntMove300,
		TravLifLDStep1TraLifNxtUnlBffr,
		TravLifLDStep1PreEntTravLifMov,
		TravLifLDStep1EntTraLifMovRotCyl,
		TravLifLDStep1USSigRechk,
		TravLifLDStep1InletPneuOpn,
		MagPlat_Step1InletPneuOpn,
		TravLifLDStep1USSigRechkTwice,
		TravLifLDStep1USMagWidthChk,
		TravLifLDStep1USComm,
		TravLifLDStep1EntPullerExt,
		TravLifLDStep1EntPullerRetWait,
		TravLifLDStep1EntTravLifMov,
		TravLifLDStep1EntBrd,
		MagPlat_Step1EntBrd,
		TravLifLDStep1InletPneuCls,
		MagPlat_Step1InletPneuCls,
		TravLifLDStep1DSSigWait,
		TravLifLDStep1ExitTravLifMov,
		TravLifLDStep1InShutClsInt,
		TravLifLDStep1DSSigRechk,
		TravLifLDStep1OutletPneuOpn,
		TravLifLDStep1DSSigRechkTwice,
		TravLifLDStep1ChkRgtSenForDBAOn,
		TravLifLDStep1DSComm,
		TravLifLDStep1ExitBrd,
		TravLifLDStep1OutletPneuCls,
		TravLifLDStep1TranInErr,
		TravLifLDStep1TranOutBrdStuckErr,
		TravLifLDStep1MagWidthErr,
		TravLifLDStep1OutletShutErr,
		TravLifLDStep1ConvEntBrdLostErr
		);
	eTravLifLDPos :
		(
		TravLifLDPosInvalid,
		TravLifLDPosUS1,
		TravLifLDPosUS2,
		TravLifLDPosUS3,
		TravLifLDPosDS1,
		TravLifLDPosDS2,
		TravLifLDPosDS3,
		TravLifLDPosUS4
		);
END_TYPE
```

### OpsTravLifLD.var - Change By Project
```iecst
(*2019-03-25*)
(**)
(*Action & State & Status*)
(**)
(*Alarm*)
VAR
	p_OpsTravLifLDAlmData : UDINT;
END_VAR
(**)
(*Output*)
VAR
	p_OpsTravLifLDStepTxt : UDINT;
	p_OpsTravLifLDPaused : UDINT;
END_VAR
(**)
VAR
	p_OpsTravLifLDUSSMEMAAct1 : UDINT;
	p_OpsTravLifLDUSSMEMAAct2 : UDINT;
	p_OpsTravLifLDUSSMEMAAct3 : UDINT;
	p_OpsTravLifLDUSSMEMAAct4 : UDINT;
	p_OpsTravLifLDDSSMEMAAct1 : UDINT;
	p_OpsTravLifLDDSSMEMAAct2 : UDINT;
	p_OpsTravLifLDDSSMEMAAct3 : UDINT;
	p_OpsTravLifLDConvAct : UDINT;
	p_OpsTravLifLDAWAct : UDINT;
	p_OpsTravLifLDAWPushPullAct : UDINT;
	p_OpsTravLifLDTravAct : UDINT;
	p_OpsTravLifLDLifAct : UDINT;
	p_OpsTravLifLDInletPneuAct : UDINT;
	p_OpsTravLifLDInletPneuAct2 : UDINT;
	p_OpsTravLifLDInletPneuAct3 : UDINT;
	p_OpsTravLifLDOutletPneuAct : UDINT;
	p_OpsTravLifLDOutletPneuAct2 : UDINT;
	p_OpsTravLifLDPullerAct : UDINT;
END_VAR
(**)
VAR
	p_OpsTravLifLDPosGo : UDINT;
	p_OpsTravLifLDMagDis : UDINT;
	p_OpsTravLifLDGoUnloadSlt1 : UDINT;
	p_OpsTravLifLDGoUnloadSlt2 : UDINT;
	p_OpsTravLifLDGoUnloadSlt3 : UDINT;
	p_OpsTravLifLDGoUnloadSlt4 : UDINT;
	p_OpsTravLifLDInitConv : UDINT;
	p_OpsTravLifLDInitDone : UDINT;
	p_OpsTravLifLDUSComm : UDINT;
	p_OpsTravLifLDEntBrd : UDINT;
	p_OpsTravLifLDDSComm : UDINT;
	p_OpsTravLifLDExitBrd : UDINT;
	p_OpsTravLifLDAWPosDiff : UDINT;
	p_OpsTravLifULInDSPos : UDINT;
	p_OpsTravLifULUpdatePullSlot : UDINT;
	p_OpsTravLifLDBypCurtainSenCtrl : UDINT;
	p_OpsTravLifLBypCurtainWidthChg : UDINT;
	p_OpsTravLifLDBypCurtainLED : UDINT;
	p_OpsTravLifLDUSMagWidthChk : UDINT;
	p_OpsTravLifULTravGotoChkPt : UDINT;
	p_OpsTravLifWChkErrCmdUnclmp1 : UDINT;
	p_OpsTravLifWChkErrCmdUnclmp2 : UDINT;
	p_OpsTravLifWChkErrCmdUnclmp3 : UDINT;
	p_OpsTravLifMove : UDINT;
	p_OpsTravLifStandby : UDINT;
END_VAR
```

### Program Logical/Operations/OpsTravLifLD (IEC) - pne

#### InputRef.var
```iecst
(*2019-04-16*)
(**)
(*General*)
VAR
	p_udiRstErr : REFERENCE TO UDINT;
	p_bEn : REFERENCE TO BOOL;
	p_bDis : REFERENCE TO BOOL;
	p_bRun : REFERENCE TO BOOL;
	p_bStop : REFERENCE TO BOOL;
	p_bStep : REFERENCE TO BOOL;
	p_bGotoStandby : REFERENCE TO BOOL;
	p_bUnlockCover : REFERENCE TO BOOL;
END_VAR
(**)
(*Configuration*)
VAR
	p_sProgNm : REFERENCE TO STRING[15];
	p_bNtSettingsLoadDone : REFERENCE TO BOOL;
END_VAR
(**)
VAR
	p_eLDMod : REFERENCE TO eLDMod;
	p_eLDMag : REFERENCE TO eLDMag;
	p_bNonBffrMod : REFERENCE TO BOOL;
	p_bUSAllow : REFERENCE TO BOOL;
	p_bDSAllow : REFERENCE TO BOOL;
	p_bPullerRotCylPrep : REFERENCE TO BOOL;
	p_diPullerExtMaxSlt : REFERENCE TO DINT;
	p_diPullerExtMinSlt : REFERENCE TO DINT;
END_VAR
(**)
VAR
	p_bProdRcpCurrRcpTopToBtm : REFERENCE TO BOOL;
	p_diProdRcpCurrRcpPitch : REFERENCE TO DINT;
	p_diProdRcpCurrRcpPitchRear : REFERENCE TO DINT;
	p_diMinSlt : REFERENCE TO DINT;
	p_diMaxSlt : REFERENCE TO DINT;
END_VAR
(**)
VAR
	p_eUSCommMod1 : REFERENCE TO eMcSetCommMod;
	p_eUSCommMod2 : REFERENCE TO eMcSetCommMod;
	p_eUSCommMod3 : REFERENCE TO eMcSetCommMod;
	p_eUSCommMod4 : REFERENCE TO eMcSetCommMod;
	p_eDSCommMod1 : REFERENCE TO eMcSetCommMod;
	p_eDSCommMod2 : REFERENCE TO eMcSetCommMod;
	p_eDSCommMod3 : REFERENCE TO eMcSetCommMod;
END_VAR
(**)
VAR
	p_eUSSMEMAStat1 : REFERENCE TO eSMEMAAction;
	p_eUSSMEMAStatus1 : REFERENCE TO eFBStatus;
	p_bUSSMEMAUSRdy1 : REFERENCE TO BOOL;
	p_bUSSMEMATransporting1 : REFERENCE TO BOOL;
	p_bUSSMEMAConvStart1 : REFERENCE TO BOOL;
	p_bUSSMEMAConvStop1 : REFERENCE TO BOOL;
END_VAR
(**)
VAR
	p_eUSSMEMAStat2 : REFERENCE TO eSMEMAAction;
	p_eUSSMEMAStatus2 : REFERENCE TO eFBStatus;
	p_bUSSMEMAUSRdy2 : REFERENCE TO BOOL;
	p_bUSSMEMATransporting2 : REFERENCE TO BOOL;
	p_bUSSMEMAConvStart2 : REFERENCE TO BOOL;
	p_bUSSMEMAConvStop2 : REFERENCE TO BOOL;
END_VAR
(**)
VAR
	p_eUSSMEMAStat3 : REFERENCE TO eSMEMAAction;
	p_eUSSMEMAStatus3 : REFERENCE TO eFBStatus;
	p_bUSSMEMAUSRdy3 : REFERENCE TO BOOL;
	p_bUSSMEMATransporting3 : REFERENCE TO BOOL;
	p_bUSSMEMAConvStart3 : REFERENCE TO BOOL;
	p_bUSSMEMAConvStop3 : REFERENCE TO BOOL;
END_VAR
(**)
VAR
	p_eUSSMEMAStat4 : REFERENCE TO eSMEMAAction;
	p_eUSSMEMAStatus4 : REFERENCE TO eFBStatus;
	p_bUSSMEMAUSRdy4 : REFERENCE TO BOOL;
	p_bUSSMEMATransporting4 : REFERENCE TO BOOL;
	p_bUSSMEMAConvStart4 : REFERENCE TO BOOL;
	p_bUSSMEMAConvStop4 : REFERENCE TO BOOL;
END_VAR
(**)
VAR
	p_eDSSMEMAStat1 : REFERENCE TO eSMEMAAction;
	p_eDSSMEMAStatus1 : REFERENCE TO eFBStatus;
	p_bDSSMEMADSRdy1 : REFERENCE TO BOOL;
	p_bDSSMEMAConvStart1 : REFERENCE TO BOOL;
END_VAR
(**)
VAR
	p_eDSSMEMAStat2 : REFERENCE TO eSMEMAAction;
	p_eDSSMEMAStatus2 : REFERENCE TO eFBStatus;
	p_bDSSMEMADSRdy2 : REFERENCE TO BOOL;
	p_bDSSMEMAConvStart2 : REFERENCE TO BOOL;
END_VAR
(**)
VAR
	p_eDSSMEMAStat3 : REFERENCE TO eSMEMAAction;
	p_eDSSMEMAStatus3 : REFERENCE TO eFBStatus;
	p_bDSSMEMADSRdy3 : REFERENCE TO BOOL;
	p_bDSSMEMAConvStart3 : REFERENCE TO BOOL;
END_VAR
(**)
VAR
	p_eDSSMEMAStat4 : REFERENCE TO eSMEMAAction;
	p_eDSSMEMAStatus4 : REFERENCE TO eFBStatus;
	p_bDSSMEMADSRdy4 : REFERENCE TO BOOL;
	p_bDSSMEMAConvStart4 : REFERENCE TO BOOL;
END_VAR
(**)
VAR
	p_bUSHermesUSRdy1 : REFERENCE TO BOOL;
	p_bUSHermesTransporting1 : REFERENCE TO BOOL;
	p_bUSHermesStopTransport1 : REFERENCE TO BOOL;
END_VAR
(**)
VAR
	p_bUSHermesUSRdy2 : REFERENCE TO BOOL;
	p_bUSHermesTransporting2 : REFERENCE TO BOOL;
	p_bUSHermesStopTransport2 : REFERENCE TO BOOL;
END_VAR
(**)
VAR
	p_bUSHermesUSRdy3 : REFERENCE TO BOOL;
	p_bUSHermesTransporting3 : REFERENCE TO BOOL;
	p_bUSHermesStopTransport3 : REFERENCE TO BOOL;
END_VAR
(**)
VAR
	p_bUSHermesUSRdy4 : REFERENCE TO BOOL;
	p_bUSHermesTransporting4 : REFERENCE TO BOOL;
	p_bUSHermesStopTransport4 : REFERENCE TO BOOL;
END_VAR
(**)
VAR
	p_bDSHermesDSRdy1 : REFERENCE TO BOOL;
	p_bDSHermesTransporting1 : REFERENCE TO BOOL;
	p_bDSHermesStopTransport1 : REFERENCE TO BOOL;
END_VAR
(**)
VAR
	p_bDSHermesDSRdy2 : REFERENCE TO BOOL;
	p_bDSHermesTransporting2 : REFERENCE TO BOOL;
	p_bDSHermesStopTransport2 : REFERENCE TO BOOL;
END_VAR
(**)
VAR
	p_bDSHermesDSRdy3 : REFERENCE TO BOOL;
	p_bDSHermesTransporting3 : REFERENCE TO BOOL;
	p_bDSHermesStopTransport3 : REFERENCE TO BOOL;
END_VAR
(**)
VAR
	p_eConvStat : REFERENCE TO eConvAction;
	p_eConvStatus : REFERENCE TO eFBStatus;
	p_eConvDir : REFERENCE TO eConvDir;
	p_bConvHvBrd : REFERENCE TO BOOL;
END_VAR
(**)
VAR
	p_eMtrPshrStat : REFERENCE TO eMtrPshrAction;
	p_eMtrPshrStatus : REFERENCE TO eFBStatus;
END_VAR
(**)
VAR
	p_eAWStat : REFERENCE TO eAWAction;
	p_eAWStatus : REFERENCE TO eFBStatus;
	p_bAWWidthPosDiff : REFERENCE TO BOOL;
END_VAR
(**)
VAR
	p_eAWPushOrPullerStat : REFERENCE TO eAWAction;
	p_eAWPushOrPullerStatus : REFERENCE TO eFBStatus;
	p_bAWPushOrPullerWidthPosDiff : REFERENCE TO BOOL;
END_VAR
(**)
VAR
	p_eTravStat : REFERENCE TO eTravAction;
	p_eTravStatus : REFERENCE TO eFBStatus;
	p_bTravAPosDiff : REFERENCE TO BOOL;
	p_bTravBPosDiff : REFERENCE TO BOOL;
	p_bTravCPosDiff : REFERENCE TO BOOL;
	p_bTravDPosDiff : REFERENCE TO BOOL;
	p_bTravEPosDiff : REFERENCE TO BOOL;
	p_bTravPosDiff : REFERENCE TO BOOL;
	p_bLifterBtmPosDiff : REFERENCE TO BOOL;
	p_bLifterAPosDiff : REFERENCE TO BOOL;
	p_bLifterBPosDiff : REFERENCE TO BOOL;
END_VAR
(**)
VAR
	p_eLifStat : REFERENCE TO eLifterAction;
	p_eLifStatus : REFERENCE TO eFBStatus;
	p_tShutterWaitTmr : REFERENCE TO TIME;
	p_bOutShutDis : REFERENCE TO BOOL;
	p_bMagWidthChkDis : REFERENCE TO BOOL;
END_VAR
(**)
VAR
	p_eInletPneuStat : REFERENCE TO ePneuAction;
	p_eInletPneuStatus : REFERENCE TO eFBStatus;
	p_bInletPneuCls : REFERENCE TO BOOL;
	p_bInShutterExtended : REFERENCE TO BOOL;
	p_bInShutterRetracted : REFERENCE TO BOOL;
	p_bInShutterOpenRS : REFERENCE TO BOOL;
END_VAR
(**)
VAR
	p_eInletPneuStat2 : REFERENCE TO ePneuAction;
	p_eInletPneuStatus2 : REFERENCE TO eFBStatus;
	p_bInletPneuCls2 : REFERENCE TO BOOL;
	p_bInShutterExtended2 : REFERENCE TO BOOL;
	p_bInShutterRetracted2 : REFERENCE TO BOOL;
	p_bInShutterOpenRS2 : REFERENCE TO BOOL;
END_VAR
(**)
VAR
	p_eInletPneuStat3 : REFERENCE TO ePneuAction;
	p_eInletPneuStatus3 : REFERENCE TO eFBStatus;
	p_bInletPneuCls3 : REFERENCE TO BOOL;
	p_bInShutterExtended3 : REFERENCE TO BOOL;
	p_bInShutterRetracted3 : REFERENCE TO BOOL;
	p_bInShutterOpenRS3 : REFERENCE TO BOOL;
END_VAR
(**)
VAR
	p_eOutletPneuStat : REFERENCE TO ePneuAction;
	p_eOutletPneuStatus : REFERENCE TO eFBStatus;
	p_eOutletPneuStat2 : REFERENCE TO ePneuAction;
	p_eOutletPneuStatus2 : REFERENCE TO eFBStatus;
	p_bOutShutterOpenRS2 : REFERENCE TO BOOL;
	p_bOutShutterOpenRS : REFERENCE TO BOOL;
	p_bOutletShutPrep : REFERENCE TO BOOL;
END_VAR
(**)
VAR
	p_ePullerStat : REFERENCE TO ePneuAction;
	p_ePullerStatus : REFERENCE TO eFBStatus;
END_VAR
(**)
(*Input*)
VAR
	p_bConvLftSen : REFERENCE TO BOOL;
	p_bConvRgtSen : REFERENCE TO BOOL;
	p_bConvClrSen : REFERENCE TO BOOL;
	p_bPullerExtSen : REFERENCE TO BOOL;
	p_bPullerRetSen : REFERENCE TO BOOL;
END_VAR
(**)
(*Magazine*)
VAR
	p_bMagTransferBrd1 : REFERENCE TO BOOL;
	p_bMagTransferBrd2 : REFERENCE TO BOOL;
	p_bMagTransferBrd3 : REFERENCE TO BOOL;
	p_bMagTransferBrd4 : REFERENCE TO BOOL;
	p_bBufferMagPresent1 : REFERENCE TO BOOL;
	p_bBufferMagPresent2 : REFERENCE TO BOOL;
	p_bBufferMagPresent3 : REFERENCE TO BOOL;
	p_bBufferMagPresent4 : REFERENCE TO BOOL;
	p_diBufferNxtUnloadSlt1 : REFERENCE TO DINT;
	p_diBufferNxtUnloadSlt2 : REFERENCE TO DINT;
	p_diBufferNxtUnloadSlt3 : REFERENCE TO DINT;
	p_diBufferNxtUnloadSlt4 : REFERENCE TO DINT;
END_VAR
(**)
VAR
	p_bDBAOnRgtSen : REFERENCE TO BOOL;
	p_eConvDirection : REFERENCE TO eConvDir;
	p_bLeftSen : REFERENCE TO BOOL;
	p_bRightSen : REFERENCE TO BOOL;
	p_bTravIsHomed : REFERENCE TO BOOL;
	p_bLifterBtmIsHomed : REFERENCE TO BOOL;
	p_diSltToSltDist : REFERENCE TO DINT;
	p_bMagWidthChkSenOn : REFERENCE TO BOOL;
END_VAR
(**)
VAR
	p_bStepMagConvLD1DSCom : REFERENCE TO BOOL;
	p_bStepMagConvLD2DSCom : REFERENCE TO BOOL;
	p_bStepMagConvLD3DSCom : REFERENCE TO BOOL;
	p_bStepMagConvLD4DSCom : REFERENCE TO BOOL;
	p_bMCLD1AGVCommRdy : REFERENCE TO BOOL;
	p_bMCLD2AGVCommRdy : REFERENCE TO BOOL;
	p_bMCLD3AGVCommRdy : REFERENCE TO BOOL;
END_VAR
(**)
VAR
	p_diNtParamPullerHeightInMM : REFERENCE TO DINT;
END_VAR
(**)
VAR
	p_bMCSelfTest : REFERENCE TO BOOL;
	p_bPullerNoRotCylStartPull : REFERENCE TO BOOL;
	p_bPullerRotHmRS : REFERENCE TO BOOL;
	p_bCurtainSenPB : REFERENCE TO BOOL;
	p_bPneuUnclmpFBDone : REFERENCE TO BOOL;
	p_siCntrPullLmt : REFERENCE TO SINT;
	p_bShutter2Prep : REFERENCE TO BOOL;
	p_bShutter3Prep : REFERENCE TO BOOL;
	p_bOutShutter2Prep : REFERENCE TO BOOL;
END_VAR
(**)
```

#### InputRef_Link.var
```iecst
(*2018-12-11*)
(**)
(*External Data*)
VAR
	p_sLinkProdRcpCurrRcp0Nm : REFERENCE TO STRING[254];
	p_sLinkProdRcpCurrRcp2Nm : REFERENCE TO STRING[254];
	p_usiLinkProdRcpCurrRcpMcMod : REFERENCE TO USINT;
	p_bLinkNtParamMagConv1Prep : REFERENCE TO USINT;
	p_bLinkNtParamMagConv2Prep : REFERENCE TO USINT;
	p_bLinkNtParamMagConv3Prep : REFERENCE TO USINT;
	p_bLinkNtParamMagConv4Prep : REFERENCE TO USINT;
	p_tyBufferStat1 : REFERENCE TO tyBffrStat;
	p_tyBufferStat2 : REFERENCE TO tyBffrStat;
	p_tyBufferStat3 : REFERENCE TO tyBffrStat;
	p_tyBufferStat4 : REFERENCE TO tyBffrStat;
	p_bLinkNtParamProjRotCylPrep : REFERENCE TO USINT;
	p_bLinkProjLifterMagPlatform : REFERENCE TO BOOL;
	p_bLinkDIPullerAntiJamSen : REFERENCE TO BOOL;
	p_bLinkProjWorkOrderOPCUA : REFERENCE TO BOOL;
	p_uiLinkUIBrdOutCntr : REFERENCE TO UINT;
	p_bLinkUIBlkTravLif : REFERENCE TO BOOL;
	p_bCurtainSenPrep : REFERENCE TO BOOL;
	p_tyDISettings : REFERENCE TO tyDigitalInputSettings;
	p_bOpsMagConvLD1UnclmpDone : REFERENCE TO BOOL;
	p_bOpsMagConvLD2UnclmpDone : REFERENCE TO BOOL;
	p_bOpsMagConvLD3UnclmpDone : REFERENCE TO BOOL;
	p_bRlsMag1 : REFERENCE TO BOOL;
	p_bRlsMag2 : REFERENCE TO BOOL;
	p_bRlsMag3 : REFERENCE TO BOOL;
	p_bEjectMag1 : REFERENCE TO BOOL;
	p_bEjectMag2 : REFERENCE TO BOOL;
	p_bEjectMag3 : REFERENCE TO BOOL;
	p_bLinkDIUnlockSafetySig : REFERENCE TO BOOL;
	p_eNtParamCustomerReq : REFERENCE TO eCustomer;
	p_diAutoRcpTravLifPitch : REFERENCE TO DINT;
	p_bLinkFollower1USAllow : REFERENCE TO BOOL;
	p_bAutoRcpTravWidthDiffBlk : REFERENCE TO BOOL;
	p_bNtParamAutoRcpPrep : REFERENCE TO BOOL;
	p_ausiSvyMagAccOrder : REFERENCE TO ARRAY[1..3] OF USINT;
	p_bHermesSvyPrep : REFERENCE TO BOOL;
	p_bMcParamHermesSvyEn : REFERENCE TO BOOL;
	p_tyAutoRcpMagRcp : REFERENCE TO ARRAY[1..4] OF tyBoardProperty;
	p_bMcParamMesRFIDEn : REFERENCE TO BOOL;
END_VAR
```

#### Local.var
```iecst
(*2019-04-16*)
(**)
(*Local Action, State & Status*)
VAR
	eStatus : eFBStatus := Idle;
	udiStatus : UDINT := 0;
END_VAR
(**)
(*Local Alarm*)
VAR
	tyAlmData : tyAlmDat;
	a_tyAlmText : ARRAY[10000..10099] OF tyAlmTxt := [(sAlmText:='Magazine Not Present While Pulling Board Out From Magazine',sRcyText:='Insert Magazine To Continue Operation.'),(sAlmText:='Traverser And Lifter Pre-Enter Position Are Invalid',sRcyText:='Reset And Resume Operation. If The Problem Persists, Please Contact Nutek For A Possible Solution.'),(sAlmText:='Traverser And Lifter Enter Position Are Invalid',sRcyText:='Reset And Resume Operation. If The Problem Persists, Please Contact Nutek For A Possible Solution.'),(sAlmText:='Conveyor Outlet Sensor Timeout Alarm',sRcyText:='Check Conveyor Outlet Sensor'),(sAlmText:='Magazine Width Detection Failed',sRcyText:='Magazine Is Not Set In Correct Width'),(sAlmText:='Puller AntiJam Sensor On',sRcyText:='Board Jam During Puller Is Retracting'),(sAlmText:='Traverser And Lifter Moving Invalid.',sRcyText:='Please Check Retracted Puller.'),(sAlmText:='Clear Sensor Interrupt Outlet Shutter Close',sRcyText:='Please Remove The Board From Clear Sensor.'),(sAlmText:='Board Lost After Conveyor complete .',sRcyText:='Outlet Sensor False triggered or Brd Lost in the middle of transfer'),(sAlmText:='Inlet And Outlet Same Time Sensing Error',sRcyText:='Please Ensure No Blockage At Inlet Sensor.'),90((0))];
END_VAR
(**)
(*Local Output*)
VAR
	sStepTxt : STRING[80];
	bPaused : BOOL;
END_VAR
(**)
VAR
	eUSSMEMAAct1 : eSMEMAAction;
	eUSSMEMAAct2 : eSMEMAAction;
	eUSSMEMAAct3 : eSMEMAAction;
	eUSSMEMAAct4 : eSMEMAAction;
	eDSSMEMAAct1 : eSMEMAAction;
	eDSSMEMAAct2 : eSMEMAAction;
	eDSSMEMAAct3 : eSMEMAAction;
	eConvAct : eConvAction;
	eAWAct : eAWAction;
	eAWPushOrPullerAct : eAWAction;
	eTravAct : eTravAction;
	eLifAct : eLifterAction;
	eInletPneuAct : ePneuAction;
	eInletPneuAct2 : ePneuAction;
	eInletPneuAct3 : ePneuAction;
	eOutletPneuAct : ePneuAction;
	eOutletPneuAct2 : ePneuAction;
	ePullerAct : ePneuAction;
	eMtrPshrAct : eMtrPshrAction;
	bInShutClo1 : BOOL;
	bInShutClo2 : BOOL;
	bInShutClo3 : BOOL;
END_VAR
(**)
VAR
	eTravLifPosGo : eTravLifLDPos;
	a_bMagDis : ARRAY[1..4] OF BOOL;
	diGoUnloadSlt1 : DINT;
	diGoUnloadSlt2 : DINT;
	diGoUnloadSlt3 : DINT;
	diGoUnloadSlt4 : DINT;
	bInitConv : BOOL;
	bOpsInitDone : BOOL;
	bUSComm : BOOL;
	bEntBrd : BOOL;
	bDSComm : BOOL;
	bExitBrd : BOOL;
	bStepAWPosDiff : BOOL;
	bUpdatePullSlot : BOOL;
	bUSMagWidthChk : BOOL;
	bTraLifMoving : BOOL;
	bStandby : BOOL;
	fbWaitTimer : TON := (PT:=T#2s);
	fbWidthChkSenOnTim : TON := (PT:=T#0ms);
	fbWidthChkSenOffTim : TON := (PT:=T#5s);
	bLifterBtmPosDiff : BOOL;
	bLifterAPosDiff : BOOL;
	bLifterBPosDiff : BOOL;
	bBypCurtainSenPB : BOOL;
	bBypCurtainSenCtrl : BOOL;
	bBypCurtainSensorPBLED : BOOL;
	fbBypCurtainPBLEDBlinkTm : TON := (IN:=FALSE,PT:=T#500ms,Q:=FALSE,ET:=0,StartTime:=0,M:=FALSE,Restart:=0);
	bBypCurtainBtnOff : BOOL;
	bMag1CheckDone : BOOL;
	bMag2CheckDone : BOOL;
	bMag3CheckDone : BOOL;
	bBypCurtainWidthChg : BOOL;
	bTravGoToChkPt : BOOL;
END_VAR
(*Step Logger*)
VAR
	bClsLog : BOOL;
	blog : BOOL;
	logStep : ARRAY[0..999] OF eTravLifLDStep1;
	logIndexStep : INT;
	eGotoOpsStepDummy : eTravLifLDStep1;
END_VAR
(**)
(*Local Input*)
VAR
	udiRstErr : UDINT := 0;
	bEn : BOOL := TRUE;
	bDis : BOOL := FALSE;
	bRun : BOOL;
	bStop : BOOL;
	bStep : BOOL;
	bGotoStandby : BOOL;
	eLDMode : eLDMod;
	eLDMagazine : eLDMag;
	bNonBffrMod : BOOL;
	bUSAllow : BOOL := TRUE;
	bDSAllow : BOOL := TRUE;
	bPullerRotCylPrep : BOOL;
	diPullerExtMaxSlt : DINT;
	diPullerExtMinSlt : DINT;
	bProdRcpCurrRcpTopToBtm : BOOL;
	diProdRcpCurrRcpPitch : DINT;
	eUSCommMod1 : eMcSetCommMod;
	eUSCommMod2 : eMcSetCommMod;
	eUSCommMod3 : eMcSetCommMod;
	eUSCommMod4 : eMcSetCommMod;
	eDSCommMod1 : eMcSetCommMod;
	eDSCommMod2 : eMcSetCommMod;
	eDSCommMod3 : eMcSetCommMod;
	eUSSMEMAStat1 : eSMEMAAction;
	eUSSMEMAStatus1 : eFBStatus;
	bUSSMEMAUSRdy1 : BOOL;
	bUSSMEMATransporting1 : BOOL;
	bUSSMEMAConvStart1 : BOOL;
	bUSSMEMAConvStop1 : BOOL;
	eUSSMEMAStat2 : eSMEMAAction;
	eUSSMEMAStatus2 : eFBStatus;
	bUSSMEMAUSRdy2 : BOOL;
	bUSSMEMATransporting2 : BOOL;
	bUSSMEMAConvStart2 : BOOL;
	bUSSMEMAConvStop2 : BOOL;
	eUSSMEMAStat3 : eSMEMAAction;
	eUSSMEMAStatus3 : eFBStatus;
	bUSSMEMAUSRdy3 : BOOL;
	bUSSMEMATransporting3 : BOOL;
	bUSSMEMAConvStart3 : BOOL;
	bUSSMEMAConvStop3 : BOOL;
	eUSSMEMAStat4 : eSMEMAAction;
	eUSSMEMAStatus4 : eFBStatus;
	bUSSMEMAUSRdy4 : BOOL;
	bUSSMEMATransporting4 : BOOL;
	bUSSMEMAConvStart4 : BOOL;
	bUSSMEMAConvStop4 : BOOL;
	eDSSMEMAStat1 : eSMEMAAction;
	eDSSMEMAStatus1 : eFBStatus;
	bDSSMEMADSRdy1 : BOOL;
	bDSSMEMAConvStart1 : BOOL;
	eDSSMEMAStat2 : eSMEMAAction;
	eDSSMEMAStatus2 : eFBStatus;
	bDSSMEMADSRdy2 : BOOL;
	bDSSMEMAConvStart2 : BOOL;
	eDSSMEMAStat3 : eSMEMAAction;
	eDSSMEMAStatus3 : eFBStatus;
	bDSSMEMADSRdy3 : BOOL;
	bDSSMEMAConvStart3 : BOOL;
	bUSHermesUSRdy1 : BOOL;
	bUSHermesTransporting1 : BOOL;
	bUSHermesStopTransport1 : BOOL;
	bUSHermesUSRdy2 : BOOL;
	bUSHermesTransporting2 : BOOL;
	bUSHermesStopTransport2 : BOOL;
	bUSHermesUSRdy3 : BOOL;
	bUSHermesTransporting3 : BOOL;
	bUSHermesStopTransport3 : BOOL;
	bUSHermesUSRdy4 : BOOL;
	bUSHermesTransporting4 : BOOL;
	bUSHermesStopTransport4 : BOOL;
	bDSHermesDSRdy1 : BOOL;
	bDSHermesTransporting1 : BOOL;
	bDSHermesStopTransport1 : BOOL;
	bDSHermesDSRdy2 : BOOL;
	bDSHermesTransporting2 : BOOL;
	bDSHermesStopTransport2 : BOOL;
	bDSHermesDSRdy3 : BOOL;
	bDSHermesTransporting3 : BOOL;
	bDSHermesStopTransport3 : BOOL;
	eConvStat : eConvAction;
	eConvStatus : eFBStatus;
	eConvDirection : eConvDir;
	bConvHvBrd : BOOL;
	eAWStat : eAWAction;
	eAWStatus : eFBStatus;
	bAWWidthPosDiff : BOOL;
	eTravStat : eTravAction;
	eTravStatus : eFBStatus;
	eLifStat : eLifterAction;
	eLifStatus : eFBStatus;
	eInletPneuStat : ePneuAction;
	eInletPneuStatus : eFBStatus;
	bInletPneuCls : BOOL;
	eOutletPneuStat : ePneuAction;
	eOutletPneuStatus : eFBStatus;
	ePullerStat : ePneuAction;
	ePullerStatus : eFBStatus;
	bConvLftSen : BOOL;
	bConvRgtSen : BOOL;
	bConvClrSen : BOOL;
	bPullerExtSen : BOOL;
	bPullerRetSen : BOOL;
	bMagTransferBrd1 : BOOL;
	bMagTransferBrd2 : BOOL;
	bMagTransferBrd3 : BOOL;
	bMagTransferBrd4 : BOOL;
	bBufferMagPresent1 : BOOL;
	bBufferMagPresent2 : BOOL;
	bBufferMagPresent3 : BOOL;
	bBufferMagPresent4 : BOOL;
	diBufferNxtUnloadSlt1 : DINT;
	diBufferNxtUnloadSlt2 : DINT;
	diBufferNxtUnloadSlt3 : DINT;
	diBufferNxtUnloadSlt4 : DINT;
	sProgNm : STRING[15] := 'Ops TravLifLD';
	bNtSettingsLoadDone : BOOL := TRUE;
	bOutShutDis : BOOL;
	bMagWidthChkDis : BOOL;
	tShutterWaitTmr : TIME := T#0S;
	eLocalInletPneuAct : ePneuAction;
	eLocalInletPneuStat : ePneuAction;
	eLocalInletPneuStatus : eFBStatus;
	bLocalInletPneuCls : BOOL;
	bLocalInShutterExtended : BOOL;
	bLocalnShutterRetracted : BOOL;
	tyLocalBufferStat : tyBffrStat;
END_VAR
(**)
(*Local*)
VAR
	bRstErr : BOOL;
	udiRstErrOld : UDINT;
	bInitDone : BOOL;
	bInitialDone : BOOL;
	eOpsStep : eTravLifLDStep := TravLifLDStepNA;
	eGotoOpsStep : eTravLifLDStep := TravLifLDStepInitConv;
	eOpsStep1 : eTravLifLDStep1 := TravLifLDStep1NA;
	eGotoOpsStep1 : eTravLifLDStep1 := TravLifLDStep1InitConv;
	eResumeStep : eTravLifLDStep1;
	tyParamTravLif : tyParamTravLifLD;
	udi : UDINT;
	udiPosAllwGo : UDINT;
	a_bPosAllwSigOn : ARRAY[1..4] OF BOOL;
	a_udiPosAllwSum : ARRAY[1..4] OF UDINT;
	bConvOutSenOn : BOOL;
	bReachedEnd : BOOL;
	bBrdOnSen : BOOL;
	bPullerHadExtended : BOOL;
END_VAR
VAR RETAIN
	bLocalUSRdy1Set : BOOL;
	bLocalUSRdy2Set : BOOL;
	bLocalUSRdy3Set : BOOL;
	bLocalUSRdy4Set : BOOL;
	bLocalDSRdy1Set : BOOL;
	bLocalDSRdy2Set : BOOL;
END_VAR
VAR
	bLocalUSRdy1 : BOOL;
	bLocalUSRdy2 : BOOL;
	bLocalUSRdy3 : BOOL;
	bLocalUSRdy4 : BOOL;
	bLocalDSRdy1 : BOOL;
	bLocalDSRdy2 : BOOL;
	bLocalDSRdy3 : BOOL;
	bSkipCloseOutletShutter : BOOL;
	bConvInSenOnSet : BOOL;
	fbUSB1offDelay : TON := (PT:=T#2s);
	fbUSB2offDelay : TON := (PT:=T#2s);
	fbUSB3offDelay : TON := (PT:=T#2s);
	fbUSB4offDelay : TON := (PT:=T#2s);
	tExitBoardTimoutErr : TON := (PT:=T#10s);
	tTravLiftInPos : TON := (PT:=T#150ms);
	bTravLifInUSPos : BOOL;
	bTravLifInDSPos : BOOL;
	bDualLaneMode : BOOL;
	bRearLaneMode : BOOL;
	diPullingPitchPos : DINT;
	diSltToSltDist : DINT;
	bWaitForDSTxBrd : DINT;
	bInShutterClo : BOOL;
	bMagWidthChked : BOOL;
	bMagWidthChk : BOOL; (*new width chk system*)
	usiMagWidthChkStep : USINT; (*new width chk system*)
	usiInitRetExtChk : USINT;
	usiLocalAccMag : USINT;
	bOutletSafeToClo : BOOL;
	bWidthChkErrCmdUnclmp1 : BOOL;
	bWidthChkErrCmdUnclmp2 : BOOL;
	bWidthChkErrCmdUnclmp3 : BOOL;
	bCmdUnclmpFlag : BOOL;
	bPneuUnclmpFBDone : BOOL;
	bShutter2Prep : BOOL;
	bShutter3Prep : BOOL;
	bOutShutter2Prep : BOOL;
	udiModuleNum : UDINT := 6051;
	a_bRlsMagBtn : ARRAY[1..3] OF BOOL;
	siCntrPullLmt : SINT := -1;
	fbCTDPullLmt : CTD;
	fb2SenTm : TON;
END_VAR
(**)
(*Reference*)
VAR
	p_eLocalUSCommMod : REFERENCE TO eMcSetCommMod;
	p_eLocalDSCommMod : REFERENCE TO eMcSetCommMod;
	p_bLocalUSRdy : REFERENCE TO BOOL;
	p_bLocalDSRdy : REFERENCE TO BOOL;
	p_eLocalUSSMEMAAct : REFERENCE TO eSMEMAAction;
	p_eLocalUSSMEMAStat : REFERENCE TO eSMEMAAction;
	p_eLocalUSSMEMAStatus : REFERENCE TO eFBStatus;
	p_bLocalUSSMEMAUSRdy : REFERENCE TO BOOL;
	p_bLocalUSSMEMATransporting : REFERENCE TO BOOL;
	p_bLocalUSSMEMAConvStart : REFERENCE TO BOOL;
	p_bLocalUSSMEMAConvStop : REFERENCE TO BOOL;
	p_eLocalDSSMEMAAct : REFERENCE TO eSMEMAAction;
	p_eLocalDSSMEMAStat : REFERENCE TO eSMEMAAction;
	p_eLocalDSSMEMAStatus : REFERENCE TO eFBStatus;
	p_bLocalDSSMEMADSRdy : REFERENCE TO BOOL;
	p_bLocalDSSMEMAConvStart : REFERENCE TO BOOL;
	p_bLocalUSHermesUSRdy : REFERENCE TO BOOL;
	p_bLocalUSHermesTransporting : REFERENCE TO BOOL;
	p_bLocalUSHermesStopTransport : REFERENCE TO BOOL;
	p_bLocalDSHermesDSRdy : REFERENCE TO BOOL;
	p_bLocalDSHermesTransporting : REFERENCE TO BOOL;
	p_bLocalDSHermesStopTransport : REFERENCE TO BOOL;
	p_eLocalInletPneuAct : REFERENCE TO ePneuAction;
	p_eLocalInletPneuStat : REFERENCE TO ePneuAction;
	p_eLocalInletPneuStatus : REFERENCE TO eFBStatus;
	p_bLocalInletPneuCls : REFERENCE TO BOOL;
	p_bLocalInShutterExtended : REFERENCE TO BOOL;
	p_bLocalnShutterRetracted : REFERENCE TO BOOL;
	p_tyLocalBufferStat : REFERENCE TO tyBffrStat;
END_VAR
```

#### Act_Alarm.st
```iecst
(** 2019-03-25 **)
ACTION Act_Alarm:

	//Error
	IF EDGEPOS(eStatus = Error) THEN

		tyAlmData.sProgNm		:= p_sProgNm;
		tyAlmData.udiCode		:= udiStatus;
		tyAlmData.eSeverity		:= AlmSeverityError;
		tyAlmData.udiRunTime	:= tyAlmData.udiRunTime + 1;
		tyAlmData.bAlm			:= TRUE;
		tyAlmData.udiModuleNum  := udiModuleNum;
		g_sOpsTravLifLDProgNm	:= p_sProgNm;

		//Get Error Message
		IF tyAlmData.udiCode < 10000 OR tyAlmData.udiCode > 10099 THEN
			tyAlmData.sAlmMsg	:= 'Unknown';
			tyAlmData.sRcyMsg	:= 'Unknown';
		ELSE
			tyAlmData.sAlmMsg	:= a_tyAlmText[tyAlmData.udiCode].sAlmText;
			tyAlmData.sRcyMsg	:= a_tyAlmText[tyAlmData.udiCode].sRcyText;
		END_IF

	ELSIF bRstErr AND (tyAlmData.udiCode <> 0) THEN

		tyAlmData.udiCode		:= 0;
		tyAlmData.eSeverity		:= AlmSeverityNA;
		tyAlmData.sAlmMsg		:= '';
		tyAlmData.sRcyMsg		:= '';
		tyAlmData.bAlm			:= FALSE;
	END_IF

END_ACTION
```

#### Act_InitGlobal.st
```iecst
(** 2019-04-16 **)
ACTION Act_InitGlobal:

	(* Always Change If Project Change *)

	//Pass Data To Link
	p_sLinkProdRcpCurrRcp0Nm ACCESS p_ProdRcpCurrRcp0Nm;
	p_sLinkProdRcpCurrRcp2Nm ACCESS p_ProdRcpCurrRcp2Nm;

	p_usiLinkProdRcpCurrRcpMcMod ACCESS p_ProdRcpCurrRcp2McMod;

	p_bLinkNtParamMagConv1Prep ACCESS p_NtParamProjMag1ConvPrep;
	p_bLinkNtParamMagConv2Prep ACCESS p_NtParamProjMag2ConvPrep;
	p_bLinkNtParamMagConv3Prep ACCESS p_NtParamProjMag3ConvPrep;
	p_bLinkNtParamMagConv4Prep ACCESS p_NtParamProjMag4ConvPrep;
	p_bLinkNtParamProjRotCylPrep ACCESS p_NtParamProjPullerRotCylPrep;

	p_bLinkProjLifterMagPlatform ACCESS p_NtParamProjLifterMagPlatform;
	p_bLinkDIPullerAntiJamSen ACCESS p_DIPullerAntiJamSen;

	p_bLinkProjWorkOrderOPCUA ACCESS p_NtParamProjWorkOrderOPCUA;
	p_uiLinkUIBrdOutCntr ACCESS p_UIBrdOutCntr;
	p_bLinkUIBlkTravLif ACCESS p_UIBlkTravLif;

	p_tyDISettings ACCESS p_NtParamDISettings;
	p_bCurtainSenPrep ACCESS p_NtParamProjCurtainSenPrep; //shutter keep on

	p_bRlsMag1 ACCESS p_UIRlsMag1;
	p_bRlsMag2 ACCESS p_UIRlsMag2;
	p_bRlsMag3 ACCESS p_UIRlsMag3;
	p_bEjectMag1 ACCESS p_UIEjectMag1;
	p_bEjectMag2 ACCESS p_UIEjectMag2;
	p_bEjectMag3 ACCESS p_UIEjectMag3;

	p_bLinkDIUnlockSafetySig ACCESS p_DIDSUnlockSafetySig;
	p_eNtParamCustomerReq ACCESS p_NtParamCustomerReq;
	p_diAutoRcpTravLifPitch ACCESS p_AutoRcpTravLifPitch;
	p_bMcParamMesRFIDEn ACCESS p_McParamMesRFIDEn;

	//Pass Data To Internal Use
	p_udiRstErr ACCESS p_RstErrReset;
	p_bRun ACCESS p_OpsRun;
	p_bStop ACCESS p_OpsStop;
	p_bStep ACCESS p_OpsStep;

	p_bOutShutDis ACCESS p_McParamOutShutterDis;
	p_tShutterWaitTmr ACCESS p_NtParamShutterWaitTmr;
	p_bMagWidthChkDis ACCESS p_McParamMagWidthChkDis;

	p_sProgNm ACCESS p_NtParamOpsTravLifLDProgNm;
	p_bNtSettingsLoadDone ACCESS p_StartupNtSettingsLoadDone;

	p_eLDMag ACCESS p_NtParamProjMag;
//	p_bUSAllow ACCESS p_Follower1USAllow;
	p_bLinkFollower1USAllow ACCESS p_Follower1USAllow;
	p_bDSAllow ACCESS p_LFFollowerDSAllow;
	p_bPullerRotCylPrep ACCESS p_NtParamProjPullerRotCylPrep;
	p_diPullerExtMaxSlt ACCESS p_NtParamProjPullerExtMaxSlt; //bprojmagmaxslt
	p_diPullerExtMinSlt ACCESS p_NtParamProjPullerExtMinSlt; //bprojmagminslt

	p_bProdRcpCurrRcpTopToBtm ACCESS p_ProdRcpCurrRcp2TopToBtm;
	p_diProdRcpCurrRcpPitch ACCESS p_ProdRcpCurrRcp2Pitch;
	p_diMinSlt ACCESS p_ProdRcpCurrRcp2MinSltValue;
	p_diMaxSlt ACCESS p_ProdRcpCurrRcp2MaxSltValue;

	p_diProdRcpCurrRcpPitchRear ACCESS p_ProdRcpCurrRcp2PitchRear;

	p_eDSCommMod1 ACCESS p_McParamDSCommAMod;
	p_eDSCommMod2 ACCESS p_McParamDSCommBMod;

	p_eUSSMEMAStat1 ACCESS p_USSMEMA1Stat;
	p_eUSSMEMAStatus1 ACCESS p_USSMEMA1Status;
	p_bUSSMEMAUSRdy1 ACCESS p_USSMEMA1USRdy;
	p_bUSSMEMATransporting1 ACCESS p_USSMEMA1Transporting;
	p_bUSSMEMAConvStart1 ACCESS p_USSMEMA1ConvStart;
	p_bUSSMEMAConvStop1 ACCESS p_USSMEMA1ConvStop;

	p_eUSSMEMAStat2 ACCESS p_USSMEMA2Stat;
	p_eUSSMEMAStatus2 ACCESS p_USSMEMA2Status;
	p_bUSSMEMAUSRdy2 ACCESS p_USSMEMA2USRdy;
	p_bUSSMEMATransporting2 ACCESS p_USSMEMA2Transporting;
	p_bUSSMEMAConvStart2 ACCESS p_USSMEMA2ConvStart;
	p_bUSSMEMAConvStop2 ACCESS p_USSMEMA2ConvStop;

	p_eUSSMEMAStat3 ACCESS p_USSMEMA3Stat;
	p_eUSSMEMAStatus3 ACCESS p_USSMEMA3Status;
	p_bUSSMEMAUSRdy3 ACCESS p_USSMEMA3USRdy;
	p_bUSSMEMATransporting3 ACCESS p_USSMEMA3Transporting;
	p_bUSSMEMAConvStart3 ACCESS p_USSMEMA3ConvStart;
	p_bUSSMEMAConvStop3 ACCESS p_USSMEMA3ConvStop;

	p_eUSSMEMAStat4 ACCESS p_USSMEMA4Stat;
	p_eUSSMEMAStatus4 ACCESS p_USSMEMA4Status;
	p_bUSSMEMAUSRdy4 ACCESS p_USSMEMA4USRdy;
	p_bUSSMEMATransporting4 ACCESS p_USSMEMA4Transporting;
	p_bUSSMEMAConvStart4 ACCESS p_USSMEMA4ConvStart;
	p_bUSSMEMAConvStop4 ACCESS p_USSMEMA4ConvStop;

	p_eDSSMEMAStat1 ACCESS p_DSSMEMAAStat;
	p_eDSSMEMAStatus1 ACCESS p_DSSMEMAAStatus;
	p_bDSSMEMADSRdy1 ACCESS p_DSSMEMAADSRdy;
	p_bDSSMEMAConvStart1 ACCESS p_DSSMEMAAConvStart;

	p_eDSSMEMAStat2 ACCESS p_DSSMEMABStat;
	p_eDSSMEMAStatus2 ACCESS p_DSSMEMABStatus;
	p_bDSSMEMADSRdy2 ACCESS p_DSSMEMABDSRdy;
	p_bDSSMEMAConvStart2 ACCESS p_DSSMEMABConvStart;

	p_bDSHermesDSRdy1 ACCESS p_DSHermesADSRdy;
	p_bDSHermesTransporting1 ACCESS p_DSHermesATransporting;
	p_bDSHermesStopTransport1 ACCESS p_DSHermesAStopTransport;

	p_bDSHermesDSRdy2 ACCESS p_DSHermesBDSRdy;
	p_bDSHermesTransporting2 ACCESS p_DSHermesBTransporting;
	p_bDSHermesStopTransport2 ACCESS p_DSHermesBStopTransport;

	p_eConvStat ACCESS p_PullConvStat;
	p_eConvStatus ACCESS p_PullConvStatus;
	p_eConvDir ACCESS p_NtParamProjConvDir;
	p_bConvHvBrd ACCESS p_PullConvHvBrd;

	p_eAWStat ACCESS p_AWOpenStat;
	p_eAWStatus ACCESS p_AWOpenStatus;
	p_bAWWidthPosDiff ACCESS p_AWOpenWidthPosDiff;

	p_eAWPushOrPullerStat ACCESS p_AWPushOrPullerStat;
	p_eAWPushOrPullerStatus ACCESS p_AWPushOrPullerStatus;
	p_bAWPushOrPullerWidthPosDiff ACCESS p_AWPushOrPullerWidthPosDiff;

	p_eTravStat ACCESS p_TravStat;
	p_eTravStatus ACCESS p_TravStatus;
	p_bTravAPosDiff ACCESS p_TravAPosDiff;
	p_bTravBPosDiff ACCESS p_TravBPosDiff;
	p_bTravCPosDiff ACCESS p_TravCPosDiff;
	p_bTravDPosDiff ACCESS p_TravDPosDiff;
	p_bTravEPosDiff ACCESS p_TravEPosDiff;
	p_bTravPosDiff ACCESS p_TravPosDiff;

//	p_eLifStat ACCESS p_LifterBtmStat;
//	p_eLifStatus ACCESS p_LifterBtmStatus;
	p_bLifterBtmPosDiff ACCESS p_LifterBtmPosDiff;
	p_bLifterAPosDiff ACCESS p_LifterBtmAPosDiff;
	p_bLifterBPosDiff ACCESS p_LifterBtmBPosDiff;

	p_eInletPneuStat ACCESS p_Pneu2SenInShutterStat;
	p_eInletPneuStatus ACCESS p_Pneu2SenInShutterStatus;
	p_bInletPneuCls ACCESS p_Pneu2SenInShutterExtended;
	p_bInShutterExtended ACCESS p_Pneu2SenInShutterExtended;
	p_bInShutterRetracted ACCESS p_Pneu2SenInShutterRetracted;
	p_bInShutterOpenRS ACCESS p_DIInShutterOpenRS;

	p_eInletPneuStat2 ACCESS p_Pneu2SenInShutterStat2;
	p_eInletPneuStatus2 ACCESS p_Pneu2SenInShutterStatus2;
	p_bInletPneuCls2 ACCESS p_Pneu2SenInShutterExtended2;
	p_bInShutterExtended2 ACCESS p_Pneu2SenInShutterExtended2;
	p_bInShutterRetracted2 ACCESS p_Pneu2SenInShutterRetracted2;
	p_bInShutterOpenRS2 ACCESS p_DIInShutterOpenRS2;

	p_eInletPneuStat3 ACCESS p_Pneu2SenInShutterStat3;
	p_eInletPneuStatus3 ACCESS p_Pneu2SenInShutterStatus3;
	p_bInletPneuCls3 ACCESS p_Pneu2SenInShutterExtended3;
	p_bInShutterExtended3 ACCESS p_Pneu2SenInShutterExtended3;
	p_bInShutterRetracted3 ACCESS p_Pneu2SenInShutterRetracted3;
	p_bInShutterOpenRS3 ACCESS p_DIInShutterOpenRS3;

	p_eOutletPneuStat ACCESS p_Pneu2SenOutShutterStat;
	p_eOutletPneuStatus ACCESS p_Pneu2SenOutShutterStatus;
	p_bOutShutterOpenRS ACCESS p_DIOutShutterOpenRS;
	p_bOutletShutPrep ACCESS p_NtParamProjOutletShutPrep;

	p_ePullerStat ACCESS p_Pneu2SenPullerStat;
	p_ePullerStatus ACCESS p_Pneu2SenPullerStatus;

	p_bConvLftSen ACCESS p_DIConvLftSen;
	p_bConvRgtSen ACCESS p_DIConvRgtSen;
	p_bConvClrSen ACCESS p_DIConvClrSen;
	p_bPullerExtSen ACCESS p_DIPullerExtRS;
	p_bPullerRetSen ACCESS p_DIPullerRetRS;

	p_bBufferMagPresent1 ACCESS p_DIMagPresentSen1;
	p_bBufferMagPresent2 ACCESS p_DIMagPresentSen2;
	p_bBufferMagPresent3 ACCESS p_DIMagPresentSen3;
	p_bBufferMagPresent4 ACCESS p_DIMagPresentSen4;
	p_diBufferNxtUnloadSlt1 ACCESS p_Buffer1NxtUnloadSlt;
	p_diBufferNxtUnloadSlt2 ACCESS p_Buffer2NxtUnloadSlt;
	p_diBufferNxtUnloadSlt3 ACCESS p_Buffer3NxtUnloadSlt;
	p_diBufferNxtUnloadSlt4 ACCESS p_Buffer4NxtUnloadSlt;

	p_bDBAOnRgtSen	ACCESS p_McParamDBAOnRgtSen;
	p_eConvDirection ACCESS p_NtParamProjConvDir;
	p_bLeftSen ACCESS p_DIConvLftSen;
	p_bRightSen ACCESS p_DIConvRgtSen;

	p_tyBufferStat1 ACCESS p_Buffer1BffrStat;
	p_tyBufferStat2 ACCESS p_Buffer2BffrStat;
	p_tyBufferStat3 ACCESS p_Buffer3BffrStat;
	p_tyBufferStat4 ACCESS p_Buffer4BffrStat;

	p_bTravIsHomed ACCESS p_TravIsHomed;
	p_bLifterBtmIsHomed ACCESS p_LifterBtmIsHomed;

	p_diSltToSltDist ACCESS p_MagRcpCurrRcpSltToSlt;
	p_bMagWidthChkSenOn ACCESS p_DIMagWidthChkSen;

	p_bStepMagConvLD1DSCom ACCESS p_OpsMagConvLD1DSCom;
	p_bStepMagConvLD2DSCom ACCESS p_OpsMagConvLD2DSCom;
	p_bStepMagConvLD3DSCom ACCESS p_OpsMagConvLD3DSCom;
	p_bStepMagConvLD4DSCom ACCESS p_OpsMagConvLD4DSCom;

	p_bMCLD1AGVCommRdy ACCESS p_OpsMagConvLD1AGVCommRdy;
	p_bMCLD2AGVCommRdy ACCESS p_OpsMagConvLD2AGVCommRdy;
	p_bMCLD3AGVCommRdy ACCESS p_OpsMagConvLD3AGVCommRdy;

	p_diNtParamPullerHeightInMM ACCESS p_NtParamPullerHeightInMM;

	p_bPullerNoRotCylStartPull ACCESS p_OpsLifMagLDBffrExitBrd;

	p_bMCSelfTest ACCESS p_DIMcSelfTest;

	p_bCurtainSenPB ACCESS p_DIBypCurtainSensorPB; //JOHN
	p_bPullerRotHmRS ACCESS p_DIPullerRotHmRS; //JOHN

	p_bOpsMagConvLD1UnclmpDone ACCESS p_OpsMagConvLD1UnclmpDone;
	p_bOpsMagConvLD2UnclmpDone ACCESS p_OpsMagConvLD2UnclmpDone;
	p_bOpsMagConvLD3UnclmpDone ACCESS p_OpsMagConvLD3UnclmpDone;
	p_bShutter2Prep ACCESS p_NtParamProjShutter2Prep;
	p_bShutter3Prep ACCESS p_NtParamProjShutter3Prep;
	p_bOutShutter2Prep ACCESS p_NtParamProjOutShutter2Prep; //outshutter 2
	p_eOutletPneuStat2 ACCESS p_Pneu2SenOutShutterStat2;
	p_eOutletPneuStatus2 ACCESS p_Pneu2SenOutShutterStatus2;
	p_bOutShutterOpenRS2 ACCESS p_DIOutShutterOpenRS2;
	p_siCntrPullLmt ACCESS p_NtParamProjCntrPullLmt;

	//AutoRcp
	p_bAutoRcpTravWidthDiffBlk ACCESS p_AutoRcpbTravWidthDiffblk;
	p_bNtParamAutoRcpPrep ACCESS p_NtParamAutoRcpPrep;
	p_ausiSvyMagAccOrder ACCESS p_SvyHermesMagAccOrder;
	p_bHermesSvyPrep ACCESS p_NtParamHermesSvyPrep; //queryWO
	p_bMcParamHermesSvyEn ACCESS p_McParamHermesSvyEn;

	p_tyAutoRcpMagRcp ACCESS p_AutoRcpMagRcp;
END_ACTION
```

#### Act_Initial.st
```iecst
(** 2019-01-20 **)
ACTION Act_Initial:

	//Initial
	fbCTDPullLmt.PV := p_siCntrPullLmt;
	fbCTDPullLmt(LOAD:= TRUE);
	fbCTDPullLmt(LOAD:= FALSE);

END_ACTION
```

#### Act_InitLocal.st
```iecst
(** 2019-04-16 **)
ACTION Act_InitLocal:

	//Input Reference Link To Local Variable
	p_udiRstErr ACCESS ADR(udiRstErr);
	p_bEn ACCESS ADR(bEn);
	p_bDis ACCESS ADR(bDis);
	p_bRun ACCESS ADR(bRun);
	p_bStop ACCESS ADR(bStop);
	p_bStep ACCESS ADR(bStep);
	p_bGotoStandby ACCESS ADR(bGotoStandby);

	p_sProgNm ACCESS ADR(sProgNm);
	p_bNtSettingsLoadDone ACCESS ADR(bNtSettingsLoadDone);
	p_bOutShutDis ACCESS ADR(bOutShutDis);
	p_bMagWidthChkDis ACCESS ADR(bMagWidthChkDis);

	p_eLDMod ACCESS ADR(eLDMode);
	p_eLDMag ACCESS ADR(eLDMagazine);
	p_bNonBffrMod ACCESS ADR(bNonBffrMod);
	p_bUSAllow ACCESS ADR(bUSAllow);
	p_bDSAllow ACCESS ADR(bDSAllow);
	p_bPullerRotCylPrep ACCESS ADR(bPullerRotCylPrep);
	p_diPullerExtMaxSlt ACCESS ADR(diPullerExtMaxSlt);
	p_diPullerExtMinSlt ACCESS ADR(diPullerExtMinSlt);

	p_bProdRcpCurrRcpTopToBtm ACCESS ADR(bProdRcpCurrRcpTopToBtm);
	p_diProdRcpCurrRcpPitch ACCESS ADR(diProdRcpCurrRcpPitch);

	p_eUSCommMod1 ACCESS ADR(eUSCommMod1);
	p_eUSCommMod2 ACCESS ADR(eUSCommMod2);
	p_eUSCommMod3 ACCESS ADR(eUSCommMod3);
	p_eUSCommMod4 ACCESS ADR(eUSCommMod4);
	p_eDSCommMod1 ACCESS ADR(eDSCommMod1);
	p_eDSCommMod2 ACCESS ADR(eDSCommMod2);
	p_eDSCommMod3 ACCESS ADR(eDSCommMod3);

	p_eUSSMEMAStat1 ACCESS ADR(eUSSMEMAStat1);
	p_eUSSMEMAStatus1 ACCESS ADR(eUSSMEMAStatus1);
	p_bUSSMEMAUSRdy1 ACCESS ADR(bUSSMEMAUSRdy1);
	p_bUSSMEMATransporting1 ACCESS ADR(bUSSMEMATransporting1);
	p_bUSSMEMAConvStart1 ACCESS ADR(bUSSMEMAConvStart1);
	p_bUSSMEMAConvStop1 ACCESS ADR(bUSSMEMAConvStop1);

	p_eUSSMEMAStat2 ACCESS ADR(eUSSMEMAStat2);
	p_eUSSMEMAStatus2 ACCESS ADR(eUSSMEMAStatus2);
	p_bUSSMEMAUSRdy2 ACCESS ADR(bUSSMEMAUSRdy2);
	p_bUSSMEMATransporting2 ACCESS ADR(bUSSMEMATransporting2);
	p_bUSSMEMAConvStart2 ACCESS ADR(bUSSMEMAConvStart2);
	p_bUSSMEMAConvStop2 ACCESS ADR(bUSSMEMAConvStop2);

	p_eUSSMEMAStat3 ACCESS ADR(eUSSMEMAStat3);
	p_eUSSMEMAStatus3 ACCESS ADR(eUSSMEMAStatus3);
	p_bUSSMEMAUSRdy3 ACCESS ADR(bUSSMEMAUSRdy3);
	p_bUSSMEMATransporting3 ACCESS ADR(bUSSMEMATransporting3);
	p_bUSSMEMAConvStart3 ACCESS ADR(bUSSMEMAConvStart3);
	p_bUSSMEMAConvStop3 ACCESS ADR(bUSSMEMAConvStop3);

	p_eUSSMEMAStat4 ACCESS ADR(eUSSMEMAStat4);
	p_eUSSMEMAStatus4 ACCESS ADR(eUSSMEMAStatus4);
	p_bUSSMEMAUSRdy4 ACCESS ADR(bUSSMEMAUSRdy4);
	p_bUSSMEMATransporting4 ACCESS ADR(bUSSMEMATransporting4);
	p_bUSSMEMAConvStart4 ACCESS ADR(bUSSMEMAConvStart4);
	p_bUSSMEMAConvStop4 ACCESS ADR(bUSSMEMAConvStop4);

	p_eDSSMEMAStat1 ACCESS ADR(eDSSMEMAStat1);
	p_eDSSMEMAStatus1 ACCESS ADR(eDSSMEMAStatus1);
	p_bDSSMEMADSRdy1 ACCESS ADR(bDSSMEMADSRdy1);
	p_bDSSMEMAConvStart1 ACCESS ADR(bDSSMEMAConvStart1);

	p_eDSSMEMAStat2 ACCESS ADR(eDSSMEMAStat2);
	p_eDSSMEMAStatus2 ACCESS ADR(eDSSMEMAStatus2);
	p_bDSSMEMADSRdy2 ACCESS ADR(bDSSMEMADSRdy2);
	p_bDSSMEMAConvStart2 ACCESS ADR(bDSSMEMAConvStart2);

	p_eDSSMEMAStat3 ACCESS ADR(eDSSMEMAStat3);
	p_eDSSMEMAStatus3 ACCESS ADR(eDSSMEMAStatus3);
	p_bDSSMEMADSRdy3 ACCESS ADR(bDSSMEMADSRdy3);
	p_bDSSMEMAConvStart3 ACCESS ADR(bDSSMEMAConvStart3);

	p_bUSHermesUSRdy1 ACCESS ADR(bUSHermesUSRdy1);
	p_bUSHermesTransporting1 ACCESS ADR(bUSHermesTransporting1);
	p_bUSHermesStopTransport1 ACCESS ADR(bUSHermesStopTransport1);

	p_bUSHermesUSRdy2 ACCESS ADR(bUSHermesUSRdy2);
	p_bUSHermesTransporting2 ACCESS ADR(bUSHermesTransporting2);
	p_bUSHermesStopTransport2 ACCESS ADR(bUSHermesStopTransport2);

	p_bUSHermesUSRdy3 ACCESS ADR(bUSHermesUSRdy3);
	p_bUSHermesTransporting3 ACCESS ADR(bUSHermesTransporting3);
	p_bUSHermesStopTransport3 ACCESS ADR(bUSHermesStopTransport3);

	p_bUSHermesUSRdy4 ACCESS ADR(bUSHermesUSRdy4);
	p_bUSHermesTransporting4 ACCESS ADR(bUSHermesTransporting4);
	p_bUSHermesStopTransport4 ACCESS ADR(bUSHermesStopTransport4);

	p_bDSHermesDSRdy1 ACCESS ADR(bDSHermesDSRdy1);
	p_bDSHermesTransporting1 ACCESS ADR(bDSHermesTransporting1);
	p_bDSHermesStopTransport1 ACCESS ADR(bDSHermesStopTransport1);

	p_bDSHermesDSRdy2 ACCESS ADR(bDSHermesDSRdy2);
	p_bDSHermesTransporting2 ACCESS ADR(bDSHermesTransporting2);
	p_bDSHermesStopTransport2 ACCESS ADR(bDSHermesStopTransport2);

	p_bDSHermesDSRdy3 ACCESS ADR(bDSHermesDSRdy3);
	p_bDSHermesTransporting3 ACCESS ADR(bDSHermesTransporting3);
	p_bDSHermesStopTransport3 ACCESS ADR(bDSHermesStopTransport3);

	p_eConvStat	ACCESS ADR(eConvStat);
	p_eConvStatus ACCESS ADR(eConvStatus);
	p_eConvDir ACCESS ADR(eConvDirection);
	p_bConvHvBrd ACCESS ADR(bConvHvBrd);

	p_eAWStat ACCESS ADR(eAWStat);
	p_eAWStatus ACCESS ADR(eAWStatus);
	p_bAWWidthPosDiff ACCESS ADR(bAWWidthPosDiff);

	p_eTravStat ACCESS ADR(eTravStat);
	p_eTravStatus ACCESS ADR(eTravStatus);

	p_eLifStat ACCESS ADR(eLifStat);
	p_eLifStatus ACCESS ADR(eLifStatus);

	p_eInletPneuStat ACCESS ADR(eInletPneuStat);
	p_eInletPneuStatus ACCESS ADR(eInletPneuStatus);
	p_bInletPneuCls ACCESS ADR(bInletPneuCls);

	p_eOutletPneuStat ACCESS ADR(eOutletPneuStat);
	p_eOutletPneuStatus ACCESS ADR(eOutletPneuStatus);

	p_ePullerStat ACCESS ADR(ePullerStat);
	p_ePullerStatus ACCESS ADR(ePullerStatus);

	p_bConvLftSen ACCESS ADR(bConvLftSen);
	p_bConvRgtSen ACCESS ADR(bConvRgtSen);
	p_bConvClrSen ACCESS ADR(bConvClrSen);
	p_bPullerExtSen ACCESS ADR(bPullerExtSen);
	p_bPullerRetSen ACCESS ADR(bPullerRetSen);

	p_bMagTransferBrd1 ACCESS ADR(bMagTransferBrd1);
	p_bMagTransferBrd2 ACCESS ADR(bMagTransferBrd2);
	p_bMagTransferBrd3 ACCESS ADR(bMagTransferBrd3);
	p_bMagTransferBrd4 ACCESS ADR(bMagTransferBrd4);
	p_bBufferMagPresent1 ACCESS ADR(bBufferMagPresent1);
	p_bBufferMagPresent2 ACCESS ADR(bBufferMagPresent2);
	p_bBufferMagPresent3 ACCESS ADR(bBufferMagPresent3);
	p_bBufferMagPresent4 ACCESS ADR(bBufferMagPresent4);
	p_diBufferNxtUnloadSlt1 ACCESS ADR(diBufferNxtUnloadSlt1);
	p_diBufferNxtUnloadSlt2 ACCESS ADR(diBufferNxtUnloadSlt2);
	p_diBufferNxtUnloadSlt3 ACCESS ADR(diBufferNxtUnloadSlt3);
	p_diBufferNxtUnloadSlt4 ACCESS ADR(diBufferNxtUnloadSlt4);

	p_tShutterWaitTmr ACCESS ADR(tShutterWaitTmr);
	p_diSltToSltDist ACCESS ADR(diSltToSltDist);

	p_eLocalInletPneuAct ACCESS ADR(eLocalInletPneuAct);
	p_eLocalInletPneuStat ACCESS ADR(eLocalInletPneuStat);
	p_eLocalInletPneuStatus ACCESS ADR(eLocalInletPneuStatus);
	p_bLocalInletPneuCls ACCESS ADR(bLocalInletPneuCls);
	p_bLocalInShutterExtended ACCESS ADR(bLocalInShutterExtended);
	p_bLocalnShutterRetracted ACCESS ADR(bLocalnShutterRetracted);
	p_tyLocalBufferStat ACCESS ADR(tyLocalBufferStat);

	p_bPneuUnclmpFBDone ACCESS ADR(bPneuUnclmpFBDone);
	p_siCntrPullLmt ACCESS ADR(siCntrPullLmt);
	p_bShutter2Prep ACCESS ADR(bShutter2Prep);
	p_bShutter3Prep ACCESS ADR(bShutter3Prep);
	p_bOutShutter2Prep ACCESS ADR(bOutShutter2Prep);

END_ACTION
```

#### Act_Link.st
```iecst
(** 2018-12-11 **)
ACTION Act_Link:
	//Standby
	p_bGotoStandby :=  p_bLinkDIUnlockSafetySig;

	p_bPneuUnclmpFBDone := p_bOpsMagConvLD1UnclmpDone OR p_bOpsMagConvLD2UnclmpDone OR p_bOpsMagConvLD3UnclmpDone;
	p_eLDMod	:= USINT_TO_UDINT(p_usiLinkProdRcpCurrRcpMcMod);

//	IF p_bLinkNtParamMagConv1Prep = TRUE THEN
		p_bMagTransferBrd1 ACCESS p_OpsMagConvLD1MagBffrAvl;
//	ELSE
//		p_bMagTransferBrd1 ACCESS p_OpsMagLD1MagBffrAvl;
//	END_IF

//	IF p_bLinkNtParamMagConv2Prep =  TRUE THEN
		p_bMagTransferBrd2 ACCESS p_OpsMagConvLD2MagBffrAvl;
//	ELSE
//		p_bMagTransferBrd2 ACCESS p_OpsMagLD2MagBffrAvl;
//	END_IF

//	IF p_bLinkNtParamMagConv3Prep = TRUE THEN
		p_bMagTransferBrd3 ACCESS p_OpsMagConvLD3MagBffrAvl;
//	ELSE
//		p_bMagTransferBrd3 ACCESS p_OpsMagLD3MagBffrAvl;
//	END_IF

//	IF p_bLinkNtParamMagConv4Prep = TRUE THEN
		p_bMagTransferBrd4 ACCESS p_OpsMagConvLD4MagBffrAvl;
//	ELSE
//		p_bMagTransferBrd4 ACCESS p_OpsMagLD4MagBffrAvl;
//	END_IF

	IF bRearLaneMode THEN
		diProdRcpCurrRcpPitch := p_diProdRcpCurrRcpPitchRear;
	ELSIF (p_eNtParamCustomerReq = Siemens AND p_bNtParamAutoRcpPrep AND p_bHermesSvyPrep AND p_bMcParamHermesSvyEn)
		OR p_eNtParamCustomerReq = We_Fabricate AND p_bMcParamMesRFIDEn THEN
		diProdRcpCurrRcpPitch := p_diAutoRcpTravLifPitch; //autorcp pitch
	ELSE
		diProdRcpCurrRcpPitch := p_diProdRcpCurrRcpPitch;
	END_IF

	//Upstream Allow
	//Disable AutoRcp
	IF p_bNtParamAutoRcpPrep AND ((p_bHermesSvyPrep AND p_bMcParamHermesSvyEn) OR (p_eNtParamCustomerReq = We_Fabricate AND p_bMcParamMesRFIDEn)) THEN
		p_bUSAllow := (*p_bUSAllow AND*) p_bAutoRcpTravWidthDiffBlk = FALSE;
	ELSE
		p_bUSAllow	:= p_bLinkFollower1USAllow (*AND p_bLinkUSHermesABlkUS = FALSE AND p_bLinkUSHermesBBlkUS = FALSE*);// AND p_bAutoRcpTravWidthDiffBlk = FALSE;// AND p_diProdRcpCurrRcp1Width = p_diProdRcpCurrRcp2Width;
	END_IF

	diPullingPitchPos := REAL_TO_DINT(40000/DINT_TO_REAL(p_diSltToSltDist));

	IF p_bLinkProjLifterMagPlatform = FALSE THEN
		p_eLifStat ACCESS p_LifterBtmStat;
		p_eLifStatus ACCESS p_LifterBtmStatus;
		p_bLifterBtmPosDiff ACCESS p_LifterBtmPosDiff;
		p_bLifterAPosDiff ACCESS p_LifterBtmAPosDiff;
		p_bLifterBPosDiff ACCESS p_LifterBtmBPosDiff;
	ELSIF p_bLinkProjLifterMagPlatform AND p_bRun THEN
		p_eLifStat ACCESS ADR(eLifAct);
		p_eLifStatus := Done; //bi-dir
		p_bLifterBtmPosDiff ACCESS ADR(bLifterBtmPosDiff);
		p_bLifterAPosDiff ACCESS ADR(bLifterAPosDiff);
		p_bLifterBPosDiff ACCESS ADR(bLifterBPosDiff);
	END_IF

//	IF p_bRun AND p_bLinkDIPullerAntiJamSen = FALSE THEN
//		eStatus		:= Error;
//		udiStatus	:= 10005;
//	END_IF

//	IF (p_eConvStatus = Done AND p_eConvStat = ConvActEntPuller)
//		THEN
//			bBrdOnSen			:= FALSE;
//			eConvAct			:= ConvActIdle;
//	END_IF

//	IF p_eInletPneuStatus = Done AND p_eInletPneuStat = PneuActExt THEN
//		eInletPneuAct	:= PneuActIdle;
//	END_IF

	//Bypass Curtain Sensor PB Pressed
	IF p_bRun THEN
		IF EDGEPOS(p_bRlsMag1 OR p_bRlsMag2 OR p_bRlsMag3 OR p_bEjectMag1 OR p_bEjectMag2 OR p_bEjectMag3) THEN
			bBypCurtainSenPB := TRUE;
			bBypCurtainSensorPBLED := TRUE;

		ELSIF EDGENEG (p_bCurtainSenPB) THEN  //DI
			IF bBypCurtainSenPB 		= TRUE THEN
				bBypCurtainSenPB		:= FALSE;
				bBypCurtainSensorPBLED	:= FALSE;
				bBypCurtainSenCtrl		:= FALSE;
			ELSE
				bBypCurtainSenPB 		:= TRUE;
				bBypCurtainSensorPBLED	:= TRUE;
			END_IF
		END_IF
	ELSE
		bBypCurtainSenPB		:= FALSE;
		bBypCurtainSensorPBLED	:= FALSE;
		bBypCurtainSenCtrl		:= FALSE;
	END_IF

	//Run & Initializing Done Bypass the Curtain Sensor
	IF p_bRun AND bOpsInitDone AND bBypCurtainSenPB THEN
		bBypCurtainSenCtrl		:= TRUE;
	ELSE
		bBypCurtainSenCtrl		:= FALSE;
	END_IF

	// BypCurtainSensorPBLED
	IF  (bBypCurtainSenPB = TRUE) AND (bBypCurtainSenCtrl = TRUE) THEN // OR (p_bMCLD1AGVCommRdy OR p_bMCLD2AGVCommRdy OR p_bMCLD3AGVCommRdy) THEN		// JOHN
		bBypCurtainSensorPBLED := TRUE;					//steady on
		fbBypCurtainPBLEDBlinkTm(IN := FALSE);
	ELSIF (bBypCurtainSenPB = TRUE) AND (bBypCurtainSenCtrl = FALSE) THEN
		fbBypCurtainPBLEDBlinkTm(IN := TRUE);
		IF fbBypCurtainPBLEDBlinkTm.Q = TRUE THEN
			fbBypCurtainPBLEDBlinkTm(IN := FALSE);
			IF bBypCurtainSensorPBLED = FALSE THEN
				bBypCurtainSensorPBLED := TRUE;
			ELSE
				bBypCurtainSensorPBLED := FALSE;
			END_IF
		END_IF
	ELSE
		bBypCurtainSensorPBLED := FALSE;
		fbBypCurtainPBLEDBlinkTm(IN := FALSE);
	END_IF

	//Release mag button
	IF p_bRlsMag1 AND eTravLifPosGo = TravLifLDPosUS1 THEN
		a_bRlsMagBtn[1] := TRUE;
	ELSIF p_bRlsMag2 AND eTravLifPosGo = TravLifLDPosUS2 THEN
		a_bRlsMagBtn[2] := TRUE;
	ELSIF p_bRlsMag3 AND eTravLifPosGo = TravLifLDPosUS3 THEN
		a_bRlsMagBtn[3] := TRUE;
	END_IF

	//Inlet and outlet sensor trigger at the same time alm
	fb2SenTm(IN:= p_bRightSen = TRUE AND p_bLeftSen= TRUE, PT:= T#500ms);
	IF fb2SenTm.Q = TRUE THEN
		eStatus := Error;
		udiStatus := 10009; //'Inlet and outlet same time sensing error'
	END_IF
END_ACTION
```

#### Init.st
```iecst
(** 2019-03-25 **)
PROGRAM _INIT

	(* Always Change If Project Change *)

	//Pass Address To Global Address For External Use
	//Action, State & Status

	//Alarm
	p_OpsTravLifLDAlmData	:= ADR(tyAlmData);

	//Output
	p_OpsTravLifLDStepTxt	:= ADR(sStepTxt);
	p_OpsTravLifLDPaused	:= ADR(bPaused);

	p_OpsTravLifLDUSSMEMAAct1	:= ADR(eUSSMEMAAct1);
	p_OpsTravLifLDUSSMEMAAct2 	:= ADR(eUSSMEMAAct2);
	p_OpsTravLifLDUSSMEMAAct3	:= ADR(eUSSMEMAAct3);
	p_OpsTravLifLDUSSMEMAAct4	:= ADR(eUSSMEMAAct4);
	p_OpsTravLifLDDSSMEMAAct1	:= ADR(eDSSMEMAAct1);
	p_OpsTravLifLDDSSMEMAAct2	:= ADR(eDSSMEMAAct2);
	p_OpsTravLifLDDSSMEMAAct3	:= ADR(eDSSMEMAAct3);
	p_OpsTravLifLDConvAct		:= ADR(eConvAct);
	p_OpsTravLifLDAWAct			:= ADR(eAWAct);
	p_OpsTravLifLDAWPushPullAct	:= ADR(eAWPushOrPullerAct);
	p_OpsTravLifLDTravAct		:= ADR(eTravAct);
	p_OpsTravLifLDLifAct		:= ADR(eLifAct);
	p_OpsTravLifLDInletPneuAct	:= ADR(eInletPneuAct);
	p_OpsTravLifLDInletPneuAct2	:= ADR(eInletPneuAct2);
	p_OpsTravLifLDInletPneuAct3	:= ADR(eInletPneuAct3);
	p_OpsTravLifLDOutletPneuAct	:= ADR(eOutletPneuAct);
	p_OpsTravLifLDOutletPneuAct2	:= ADR(eOutletPneuAct2);
	p_OpsTravLifLDPullerAct		:= ADR(ePullerAct);

	p_OpsTravLifLDPosGo			:= ADR(eTravLifPosGo);
	p_OpsTravLifLDMagDis		:= ADR(a_bMagDis);
	p_OpsTravLifLDGoUnloadSlt1	:= ADR(diGoUnloadSlt1);
	p_OpsTravLifLDGoUnloadSlt2	:= ADR(diGoUnloadSlt2);
	p_OpsTravLifLDGoUnloadSlt3	:= ADR(diGoUnloadSlt3);
	p_OpsTravLifLDGoUnloadSlt4	:= ADR(diGoUnloadSlt4);

	p_OpsTravLifLDInitConv		:= ADR(bInitConv);
	p_OpsTravLifLDInitDone		:= ADR(bOpsInitDone);
	p_OpsTravLifLDUSComm		:= ADR(bUSComm);
	p_OpsTravLifLDEntBrd		:= ADR(bEntBrd);
	p_OpsTravLifLDDSComm		:= ADR(bDSComm);
	p_OpsTravLifLDExitBrd		:= ADR(bExitBrd);
	p_OpsTravLifLDAWPosDiff		:= ADR(bStepAWPosDiff);
	p_OpsTravLifULInDSPos		:= ADR(bTravLifInDSPos);
	p_OpsTravLifULUpdatePullSlot		:= ADR(	bUpdatePullSlot);
	p_OpsTravLifLDBypCurtainLED 		:= ADR (bBypCurtainSensorPBLED); 	//JOHN
	p_OpsTravLifLDBypCurtainSenCtrl		:= ADR (bBypCurtainSenCtrl); 				//JOHN
	p_OpsTravLifLBypCurtainWidthChg 	:= ADR (bBypCurtainWidthChg);

	p_OpsTravLifLDUSMagWidthChk 	:= ADR(bUSMagWidthChk);
	p_OpsTravLifULTravGotoChkPt			:= ADR (bTravGoToChkPt);

	p_OpsTravLifWChkErrCmdUnclmp1		:= ADR (bWidthChkErrCmdUnclmp1); //to opsmagconvLD1,2,3
	p_OpsTravLifWChkErrCmdUnclmp2		:= ADR (bWidthChkErrCmdUnclmp2);
	p_OpsTravLifWChkErrCmdUnclmp3		:= ADR (bWidthChkErrCmdUnclmp3);
	p_OpsTravLifMove				 	:= ADR (bTraLifMoving);
	p_OpsTravLifStandby					:= ADR(bStandby);

	(* Always Change If Project Change *)

END_PROGRAM
```

#### Act_OpsInitial.st - Do Not Change!!!
```iecst
(** 2019-01-16 **)
ACTION Act_OpsInitial:

	eOpsStep		:= TravLifLDStepNA;
	eGotoOpsStep	:= TravLifLDStepInitConv;

	eOpsStep1		:= TravLifLDStep1NA;
	eGotoOpsStep1	:= TravLifLDStep1InitConv;

	bInitConv		:= FALSE;
	bOpsInitDone	:= FALSE;
	bUSComm			:= FALSE;
	bEntBrd			:= FALSE;
	bDSComm			:= FALSE;
	bExitBrd		:= FALSE;

	bTravGoToChkPt := FALSE;

	bInShutClo1	:= FALSE;
	bInShutClo2 := FALSE;
	bInShutClo3 := FALSE;
END_ACTION
```

#### Act_OpsCommSig.st
```iecst
ACTION Act_OpsCommSig:

	//Upstream
	IF p_eUSCommMod1 = McSetCommModHermes THEN
		bLocalUSRdy1	:= p_bUSHermesUSRdy1;
	ELSE
		bLocalUSRdy1	:= p_bUSSMEMAUSRdy1;
	END_IF

	IF p_eUSCommMod2 = McSetCommModHermes THEN
		bLocalUSRdy2	:= p_bUSHermesUSRdy2;
	ELSE
		bLocalUSRdy2	:= p_bUSSMEMAUSRdy2;
	END_IF

	IF p_eUSCommMod3 = McSetCommModHermes THEN
		bLocalUSRdy3	:= p_bUSHermesUSRdy3;
	ELSE
		bLocalUSRdy3	:= p_bUSSMEMAUSRdy3;
	END_IF

	IF p_eUSCommMod4 = McSetCommModHermes THEN
		bLocalUSRdy4	:= p_bUSHermesUSRdy4;
	ELSE
		bLocalUSRdy4	:= p_bUSSMEMAUSRdy4;
	END_IF

	IF bDualLaneMode = FALSE THEN

			IF bLocalUSRdy1 AND bLocalUSRdy2Set = FALSE AND bLocalUSRdy3Set = FALSE AND bLocalUSRdy4Set = FALSE THEN
				bLocalUSRdy1Set := TRUE;
			ELSIF bLocalUSRdy1 AND bLocalUSRdy2 AND bLocalUSRdy1Set AND bLocalUSRdy2Set = FALSE THEN
				bLocalUSRdy1Set := TRUE;
			ELSIF bLocalUSRdy1 AND bLocalUSRdy3 AND bLocalUSRdy1Set AND bLocalUSRdy3Set = FALSE THEN
				bLocalUSRdy1Set := TRUE;
			ELSIF bLocalUSRdy1 AND bLocalUSRdy4 AND bLocalUSRdy1Set AND bLocalUSRdy4Set = FALSE THEN
				bLocalUSRdy1Set := TRUE;
			ELSIF p_bBufferMagPresent1 = FALSE THEN
				bLocalUSRdy1Set := FALSE;
			END_IF

			IF bLocalUSRdy2 AND bLocalUSRdy1Set = FALSE AND bLocalUSRdy3Set = FALSE AND bLocalUSRdy4Set = FALSE THEN
				bLocalUSRdy2Set := TRUE;
			ELSIF bLocalUSRdy2 AND bLocalUSRdy1 AND bLocalUSRdy2Set AND bLocalUSRdy1Set = FALSE THEN
				bLocalUSRdy2Set := TRUE;
			ELSIF bLocalUSRdy2 AND bLocalUSRdy3 AND bLocalUSRdy2Set AND bLocalUSRdy3Set = FALSE THEN
				bLocalUSRdy2Set := TRUE;
			ELSIF bLocalUSRdy2 AND bLocalUSRdy4 AND bLocalUSRdy2Set AND bLocalUSRdy4Set = FALSE THEN
				bLocalUSRdy4Set := TRUE;
			ELSIF p_bBufferMagPresent2 = FALSE THEN
				bLocalUSRdy2Set := FALSE;
			END_IF

			IF bLocalUSRdy3 AND bLocalUSRdy1Set = FALSE AND bLocalUSRdy2Set = FALSE  AND bLocalUSRdy4Set = FALSE THEN
				bLocalUSRdy3Set := TRUE;
			ELSIF bLocalUSRdy3 AND bLocalUSRdy1 AND bLocalUSRdy3Set AND bLocalUSRdy1Set = FALSE THEN
				bLocalUSRdy3Set := TRUE;
			ELSIF bLocalUSRdy3 AND bLocalUSRdy2 AND bLocalUSRdy3Set AND bLocalUSRdy2Set = FALSE THEN
				bLocalUSRdy3Set := TRUE;
			ELSIF bLocalUSRdy3 AND bLocalUSRdy4 AND bLocalUSRdy3Set AND bLocalUSRdy4Set = FALSE THEN
				bLocalUSRdy3Set := TRUE;
			ELSIF p_bBufferMagPresent3 = FALSE THEN
				bLocalUSRdy3Set := FALSE;
			END_IF

			IF bLocalUSRdy4 AND bLocalUSRdy1Set = FALSE AND bLocalUSRdy2Set = FALSE  AND bLocalUSRdy3Set = FALSE THEN
				bLocalUSRdy4Set := TRUE;
			ELSIF bLocalUSRdy4 AND bLocalUSRdy1 AND bLocalUSRdy4Set AND bLocalUSRdy1Set = FALSE THEN
				bLocalUSRdy4Set := TRUE;
			ELSIF bLocalUSRdy4 AND bLocalUSRdy2 AND bLocalUSRdy4Set AND bLocalUSRdy2Set = FALSE THEN
				bLocalUSRdy4Set := TRUE;
			ELSIF bLocalUSRdy4 AND bLocalUSRdy3 AND bLocalUSRdy4Set AND bLocalUSRdy3Set = FALSE THEN
				bLocalUSRdy4Set := TRUE;
			ELSIF p_bBufferMagPresent4 = FALSE THEN
				bLocalUSRdy4Set := FALSE;
			END_IF

	ELSE

		IF bLocalUSRdy1 AND bLocalUSRdy2Set = FALSE THEN
			bLocalUSRdy1Set := TRUE;
		ELSIF bLocalUSRdy1 AND bLocalUSRdy2 AND bLocalUSRdy1Set AND bLocalUSRdy2Set = FALSE THEN
			bLocalUSRdy1Set := TRUE;
		ELSIF p_bBufferMagPresent1 = FALSE THEN
			bLocalUSRdy1Set := FALSE;
		END_IF

		IF bLocalUSRdy2 AND bLocalUSRdy1Set = FALSE THEN
			bLocalUSRdy2Set := TRUE;
		ELSIF bLocalUSRdy2 AND bLocalUSRdy1 AND bLocalUSRdy2Set AND bLocalUSRdy1Set = FALSE THEN
			bLocalUSRdy2Set := TRUE;
		ELSIF p_bBufferMagPresent2 = FALSE THEN
			bLocalUSRdy2Set := FALSE;
		END_IF

		IF bLocalUSRdy3 AND  bLocalUSRdy4Set = FALSE THEN
			bLocalUSRdy3Set := TRUE;
		ELSIF bLocalUSRdy3 AND bLocalUSRdy4 AND bLocalUSRdy3Set AND bLocalUSRdy4Set = FALSE THEN
			bLocalUSRdy3Set := TRUE;
		ELSIF p_bBufferMagPresent3 = FALSE THEN
			bLocalUSRdy3Set := FALSE;
		END_IF

		IF bLocalUSRdy4 AND bLocalUSRdy3Set = FALSE THEN
			bLocalUSRdy4Set := TRUE;
		ELSIF bLocalUSRdy4 AND bLocalUSRdy3 AND bLocalUSRdy4Set AND bLocalUSRdy3Set = FALSE THEN
			bLocalUSRdy4Set := TRUE;
		ELSIF p_bBufferMagPresent4 = FALSE THEN
			bLocalUSRdy4Set := FALSE;
		END_IF
	END_IF

	//Downstream
	IF p_eDSCommMod1 = McSetCommModHermes THEN
		bLocalDSRdy1	:= p_bDSHermesDSRdy1;
	ELSE
		bLocalDSRdy1	:= p_bDSSMEMADSRdy1;
	END_IF

	IF p_eDSCommMod2 = McSetCommModHermes THEN
		bLocalDSRdy2	:= p_bDSHermesDSRdy2;
	ELSE
		bLocalDSRdy2	:= p_bDSSMEMADSRdy2;
	END_IF

	IF p_eDSCommMod3 = McSetCommModHermes THEN
		bLocalDSRdy3	:= p_bDSHermesDSRdy3;
	ELSE
		bLocalDSRdy3	:= p_bDSSMEMADSRdy3;
	END_IF

END_ACTION
```
